ABB RAPID module: Module1.mod

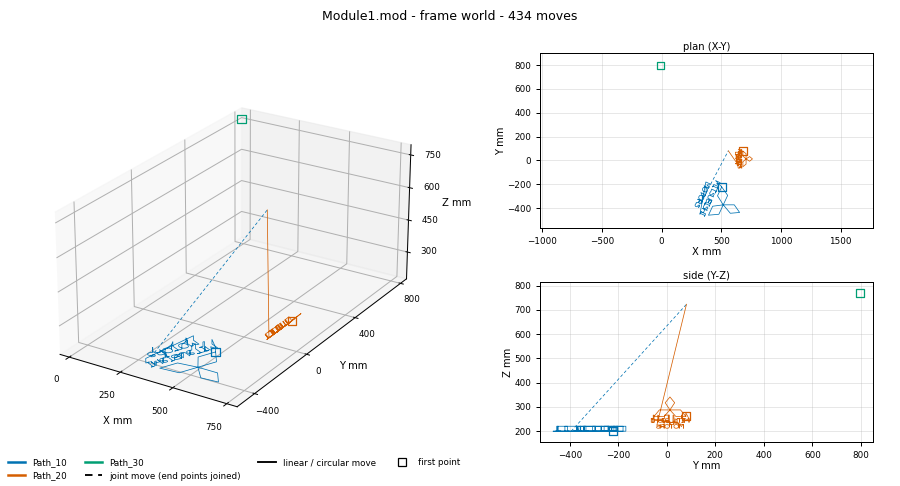
[picture p0: tool path of Module1.mod in frame world, 434 of 434 moves have a stored position in this frame; points joined in program order, loops and branches not executed]
MODULE Module1
    PERS tooldata TCP:=[TRUE,[[-35.118,-0.77,114.286],[1,0,0,0]],[1,[0,0,1],[1,0,0,0],0,0,0]];
    TASK PERS wobjdata Workobject_5:=[FALSE,TRUE,"",[[411.94279579,7.766562071,169.6],[0.537299678,0,0,-0.843391401]],[[0,0,30],[1,0,0,0]]];
    TASK PERS wobjdata Workobject_6:=[FALSE,TRUE,"",[[628.009,163.117,186.516],[0.653281027,0.27059915,-0.27059915,-0.653281027]],[[0,0,15],[1,0,0,0]]];

    CONST robtarget Target_4030:=[[169.057210378,179.421981942,0],[0,0.923879533,-0.382683432,0],[0, 0, 0, 0],[9E+09,9E+09,9E+09,9E+09,9E+09,9E+09]];
    CONST robtarget Target_4040:=[[212.704790581,255.022303499,0],[0,0.923879533,-0.382683432,0],[0, 0, 0, 0],[9E+09,9E+09,9E+09,9E+09,9E+09,9E+09]];
    CONST robtarget Target_4050:=[[387.295111711,255.022303682,0],[0,0.923879533,-0.382683432,0],[0, 0, 0, 0],[9E+09,9E+09,9E+09,9E+09,9E+09,9E+09]];
    CONST robtarget Target_4060:=[[430.942692072,179.421982217,0],[0,0.923879533,-0.382683432,0],[0, 0, 0, 0],[9E+09,9E+09,9E+09,9E+09,9E+09,9E+09]];
    CONST robtarget Target_4070:=[[348.163115412,179.42198213,0],[0,0.923879533,-0.382683432,0],[0, 0, 0, 0],[9E+09,9E+09,9E+09,9E+09,9E+09,9E+09]];
    CONST robtarget Target_4080:=[[299.999951146,255.02230359,0],[0,0.923879533,-0.382683432,0],[0, 0, 0, 0],[9E+09,9E+09,9E+09,9E+09,9E+09,9E+09]];
    CONST robtarget Target_4090:=[[260.995941008,338.665964696,0],[0,0.923879533,-0.382683432,0],[0, 0, 0, 0],[9E+09,9E+09,9E+09,9E+09,9E+09,9E+09]];
    CONST robtarget Target_4100:=[[299.999950987,406.221532398,0],[0,0.923879533,-0.382683432,0],[0, 0, 0, 0],[9E+09,9E+09,9E+09,9E+09,9E+09,9E+09]];
    CONST robtarget Target_4110:=[[339.003961108,338.665964778,0],[0,0.923879533,-0.382683432,0],[0, 0, 0, 0],[9E+09,9E+09,9E+09,9E+09,9E+09,9E+09]];
    CONST robtarget Target_4120:=[[299.999951146,255.02230359,0],[0,0.923879533,-0.382683432,0],[0, 0, 0, 0],[9E+09,9E+09,9E+09,9E+09,9E+09,9E+09]];
    CONST robtarget Target_4130:=[[251.837494145,179.422689136,0],[0,0.923879533,-0.382683432,0],[0, 0, 0, 0],[9E+09,9E+09,9E+09,9E+09,9E+09,9E+09]];
    CONST robtarget Target_4140:=[[169.057210378,179.421981942,0],[0,0.923879533,-0.382683432,0],[0, 0, 0, 0],[9E+09,9E+09,9E+09,9E+09,9E+09,9E+09]];
    CONST robtarget Target_4150:=[[169.057210378,179.421981942,20.4],[0,0.923879533,-0.382683432,0],[0, 0, 0, 0],[9E+09,9E+09,9E+09,9E+09,9E+09,9E+09]];
    CONST robtarget Target_4160:=[[142.914058536,110.942932798,20.4],[0,0.923879533,-0.382683432,0],[0, 0, 0, 0],[9E+09,9E+09,9E+09,9E+09,9E+09,9E+09]];
    CONST robtarget Target_4170:=[[142.914058536,110.942932798,0],[0,0.923879533,-0.382683432,0],[0, 0, 0, 0],[9E+09,9E+09,9E+09,9E+09,9E+09,9E+09]];
    CONST robtarget Target_4180:=[[142.914058492,152.942247173,0],[0,0.923879533,-0.382683432,0],[0, 0, 0, 0],[9E+09,9E+09,9E+09,9E+09,9E+09,9E+09]];
    CONST robtarget Target_4190:=[[150.538083807,152.942247181,0],[0,0.923879533,-0.382683432,0],[0, 0, 0, 0],[9E+09,9E+09,9E+09,9E+09,9E+09,9E+09]];
    CONST robtarget Target_4200:=[[161.020941862,129.560347259,0],[0,0.923879533,-0.382683432,0],[0, 0, 0, 0],[9E+09,9E+09,9E+09,9E+09,9E+09,9E+09]];
    CONST robtarget Target_4210:=[[171.163681507,152.942954309,0],[0,0.923879533,-0.382683432,0],[0, 0, 0, 0],[9E+09,9E+09,9E+09,9E+09,9E+09,9E+09]];
    CONST robtarget Target_4220:=[[178.923471324,152.942954318,0],[0,0.923879533,-0.382683432,0],[0, 0, 0, 0],[9E+09,9E+09,9E+09,9E+09,9E+09,9E+09]];
    CONST robtarget Target_4230:=[[178.923471368,110.942225729,0],[0,0.923879533,-0.382683432,0],[0, 0, 0, 0],[9E+09,9E+09,9E+09,9E+09,9E+09,9E+09]];
    CONST robtarget Target_4240:=[[178.923471368,110.942225729,20.4],[0,0.923879533,-0.382683432,0],[0, 0, 0, 0],[9E+09,9E+09,9E+09,9E+09,9E+09,9E+09]];
    CONST robtarget Target_4250:=[[185.798670601,110.942932843,20.4],[0,0.923879533,-0.382683432,0],[0, 0, 0, 0],[9E+09,9E+09,9E+09,9E+09,9E+09,9E+09]];
    CONST robtarget Target_4260:=[[185.798670601,110.942932843,0],[0,0.923879533,-0.382683432,0],[0, 0, 0, 0],[9E+09,9E+09,9E+09,9E+09,9E+09,9E+09]];
    CONST robtarget Target_4270:=[[202.067783423,110.94293286,0],[0,0.923879533,-0.382683432,0],[0, 0, 0, 0],[9E+09,9E+09,9E+09,9E+09,9E+09,9E+09]];
    CONST robtarget Target_4280:=[[193.933227012,110.942932851,0],[0,0.923879533,-0.382683432,0],[0, 0, 0, 0],[9E+09,9E+09,9E+09,9E+09,9E+09,9E+09]];
    CONST robtarget Target_4290:=[[193.933226968,152.942247227,0],[0,0.923879533,-0.382683432,0],[0, 0, 0, 0],[9E+09,9E+09,9E+09,9E+09,9E+09,9E+09]];
    CONST robtarget Target_4300:=[[185.798670557,152.942247218,0],[0,0.923879533,-0.382683432,0],[0, 0, 0, 0],[9E+09,9E+09,9E+09,9E+09,9E+09,9E+09]];
    CONST robtarget Target_4310:=[[202.067783379,152.942247235,0],[0,0.923879533,-0.382683432,0],[0, 0, 0, 0],[9E+09,9E+09,9E+09,9E+09,9E+09,9E+09]];
    CONST robtarget Target_4320:=[[202.067783379,152.942247235,20.4],[0,0.923879533,-0.382683432,0],[0, 0, 0, 0],[9E+09,9E+09,9E+09,9E+09,9E+09,9E+09]];
    CONST robtarget Target_4330:=[[204.689028217,152.942954345,20.4],[0,0.923879533,-0.382683432,0],[0, 0, 0, 0],[9E+09,9E+09,9E+09,9E+09,9E+09,9E+09]];
    CONST robtarget Target_4340:=[[204.689028217,152.942954345,0],[0,0.923879533,-0.382683432,0],[0, 0, 0, 0],[9E+09,9E+09,9E+09,9E+09,9E+09,9E+09]];
    CONST robtarget Target_4350:=[[238.451962805,152.94295438,0],[0,0.923879533,-0.382683432,0],[0, 0, 0, 0],[9E+09,9E+09,9E+09,9E+09,9E+09,9E+09]];
    CONST robtarget Target_4360:=[[221.570495511,152.942954362,0],[0,0.923879533,-0.382683432,0],[0, 0, 0, 0],[9E+09,9E+09,9E+09,9E+09,9E+09,9E+09]];
    CONST robtarget Target_4370:=[[221.570495555,110.942225773,0],[0,0.923879533,-0.382683432,0],[0, 0, 0, 0],[9E+09,9E+09,9E+09,9E+09,9E+09,9E+09]];
    CONST robtarget Target_4380:=[[221.570495555,110.942225773,20.4],[0,0.923879533,-0.382683432,0],[0, 0, 0, 0],[9E+09,9E+09,9E+09,9E+09,9E+09,9E+09]];
    CONST robtarget Target_4390:=[[240.630558839,113.461647255,20.4],[0,0.923879533,-0.382683432,0],[0, 0, 0, 0],[9E+09,9E+09,9E+09,9E+09,9E+09,9E+09]];
    CONST robtarget Target_4400:=[[240.630558839,113.461647255,0],[0,0.923879533,-0.382683432,0],[0, 0, 0, 0],[9E+09,9E+09,9E+09,9E+09,9E+09,9E+09]];
    CONST robtarget Target_4410:=[[254.414898435,110.193399727,0],[0,0.923879533,-0.382683432,0],[0, 0, 0, 0],[9E+09,9E+09,9E+09,9E+09,9E+09,9E+09]];
    CONST robtarget Target_4420:=[[260.813507697,111.181227907,0],[0,0.923879533,-0.382683432,0],[0, 0, 0, 0],[9E+09,9E+09,9E+09,9E+09,9E+09,9E+09]];
    CONST robtarget Target_4430:=[[265.374346433,114.005412395,0],[0,0.923879533,-0.382683432,0],[0, 0, 0, 0],[9E+09,9E+09,9E+09,9E+09,9E+09,9E+09]];
    CONST robtarget Target_4440:=[[268.182267456,118.056427148,0],[0,0.923879533,-0.382683432,0],[0, 0, 0, 0],[9E+09,9E+09,9E+09,9E+09,9E+09,9E+09]];
    CONST robtarget Target_4450:=[[269.186359081,122.922736017,0],[0,0.923879533,-0.382683432,0],[0, 0, 0, 0],[9E+09,9E+09,9E+09,9E+09,9E+09,9E+09]];
    CONST robtarget Target_4460:=[[267.178175815,129.508728575,0],[0,0.923879533,-0.382683432,0],[0, 0, 0, 0],[9E+09,9E+09,9E+09,9E+09,9E+09,9E+09]];
    CONST robtarget Target_4470:=[[260.847448799,133.508831629,0],[0,0.923879533,-0.382683432,0],[0, 0, 0, 0],[9E+09,9E+09,9E+09,9E+09,9E+09,9E+09]];
    CONST robtarget Target_4480:=[[256.575816733,134.631010087,0],[0,0.923879533,-0.382683432,0],[0, 0, 0, 0],[9E+09,9E+09,9E+09,9E+09,9E+09,9E+09]];
    CONST robtarget Target_4490:=[[252.236302415,135.720661632,0],[0,0.923879533,-0.382683432,0],[0, 0, 0, 0],[9E+09,9E+09,9E+09,9E+09,9E+09,9E+09]];
    CONST robtarget Target_4500:=[[248.169731314,138.01805156,0],[0,0.923879533,-0.382683432,0],[0, 0, 0, 0],[9E+09,9E+09,9E+09,9E+09,9E+09,9E+09]];
    CONST robtarget Target_4510:=[[246.756931961,142.255035391,0],[0,0.923879533,-0.382683432,0],[0, 0, 0, 0],[9E+09,9E+09,9E+09,9E+09,9E+09,9E+09]];
    CONST robtarget Target_4520:=[[249.156145265,147.037198555,0],[0,0.923879533,-0.382683432,0],[0, 0, 0, 0],[9E+09,9E+09,9E+09,9E+09,9E+09,9E+09]];
    CONST robtarget Target_4530:=[[255.435960587,148.857998523,0],[0,0.923879533,-0.382683432,0],[0, 0, 0, 0],[9E+09,9E+09,9E+09,9E+09,9E+09,9E+09]];
    CONST robtarget Target_4540:=[[262.004275478,147.496817976,0],[0,0.923879533,-0.382683432,0],[0, 0, 0, 0],[9E+09,9E+09,9E+09,9E+09,9E+09,9E+09]];
    CONST robtarget Target_4550:=[[267.144234674,144.297159797,0],[0,0.923879533,-0.382683432,0],[0, 0, 0, 0],[9E+09,9E+09,9E+09,9E+09,9E+09,9E+09]];
    CONST robtarget Target_4560:=[[267.144234674,144.297159797,20.4],[0,0.923879533,-0.382683432,0],[0, 0, 0, 0],[9E+09,9E+09,9E+09,9E+09,9E+09,9E+09]];
    CONST robtarget Target_4570:=[[274.35955226,152.942247311,20.4],[0,0.923879533,-0.382683432,0],[0, 0, 0, 0],[9E+09,9E+09,9E+09,9E+09,9E+09,9E+09]];
    CONST robtarget Target_4580:=[[274.35955226,152.942247311,0],[0,0.923879533,-0.382683432,0],[0, 0, 0, 0],[9E+09,9E+09,9E+09,9E+09,9E+09,9E+09]];
    CONST robtarget Target_4590:=[[274.360259381,139.838851549,0],[0,0.923879533,-0.382683432,0],[0, 0, 0, 0],[9E+09,9E+09,9E+09,9E+09,9E+09,9E+09]];
    CONST robtarget Target_4600:=[[274.359552288,126.735455787,0],[0,0.923879533,-0.382683432,0],[0, 0, 0, 0],[9E+09,9E+09,9E+09,9E+09,9E+09,9E+09]];
    CONST robtarget Target_4610:=[[275.261820549,119.179312724,0],[0,0.923879533,-0.382683432,0],[0, 0, 0, 0],[9E+09,9E+09,9E+09,9E+09,9E+09,9E+09]];
    CONST robtarget Target_4620:=[[278.375918818,113.938237265,0],[0,0.923879533,-0.382683432,0],[0, 0, 0, 0],[9E+09,9E+09,9E+09,9E+09,9E+09,9E+09]];
    CONST robtarget Target_4630:=[[283.072522062,111.027785758,0],[0,0.923879533,-0.382683432,0],[0, 0, 0, 0],[9E+09,9E+09,9E+09,9E+09,9E+09,9E+09]];
    CONST robtarget Target_4640:=[[289.539720684,110.057635261,0],[0,0.923879533,-0.382683432,0],[0, 0, 0, 0],[9E+09,9E+09,9E+09,9E+09,9E+09,9E+09]];
    CONST robtarget Target_4650:=[[296.074801555,111.010815209,0],[0,0.923879533,-0.382683432,0],[0, 0, 0, 0],[9E+09,9E+09,9E+09,9E+09,9E+09,9E+09]];
    CONST robtarget Target_4660:=[[300.737463667,113.938237288,0],[0,0.923879533,-0.382683432,0],[0, 0, 0, 0],[9E+09,9E+09,9E+09,9E+09,9E+09,9E+09]];
    CONST robtarget Target_4670:=[[303.868532488,119.213253879,0],[0,0.923879533,-0.382683432,0],[0, 0, 0, 0],[9E+09,9E+09,9E+09,9E+09,9E+09,9E+09]];
    CONST robtarget Target_4680:=[[304.75383017,126.735455818,0],[0,0.923879533,-0.382683432,0],[0, 0, 0, 0],[9E+09,9E+09,9E+09,9E+09,9E+09,9E+09]];
    CONST robtarget Target_4690:=[[304.75312305,139.838851581,0],[0,0.923879533,-0.382683432,0],[0, 0, 0, 0],[9E+09,9E+09,9E+09,9E+09,9E+09,9E+09]];
    CONST robtarget Target_4700:=[[304.753830143,152.942247343,0],[0,0.923879533,-0.382683432,0],[0, 0, 0, 0],[9E+09,9E+09,9E+09,9E+09,9E+09,9E+09]];
    CONST robtarget Target_4710:=[[304.753830143,152.942247343,20.4],[0,0.923879533,-0.382683432,0],[0, 0, 0, 0],[9E+09,9E+09,9E+09,9E+09,9E+09,9E+09]];
    CONST robtarget Target_4720:=[[312.751914945,152.942954458,20.4],[0,0.923879533,-0.382683432,0],[0, 0, 0, 0],[9E+09,9E+09,9E+09,9E+09,9E+09,9E+09]];
    CONST robtarget Target_4730:=[[312.751914945,152.942954458,0],[0,0.923879533,-0.382683432,0],[0, 0, 0, 0],[9E+09,9E+09,9E+09,9E+09,9E+09,9E+09]];
    CONST robtarget Target_4740:=[[312.751914989,110.942225869,0],[0,0.923879533,-0.382683432,0],[0, 0, 0, 0],[9E+09,9E+09,9E+09,9E+09,9E+09,9E+09]];
    CONST robtarget Target_4750:=[[318.776464765,110.942225875,0],[0,0.923879533,-0.382683432,0],[0, 0, 0, 0],[9E+09,9E+09,9E+09,9E+09,9E+09,9E+09]];
    CONST robtarget Target_4760:=[[324.800307434,110.942932988,0],[0,0.923879533,-0.382683432,0],[0, 0, 0, 0],[9E+09,9E+09,9E+09,9E+09,9E+09,9E+09]];
    CONST robtarget Target_4770:=[[331.795007712,111.724993096,0],[0,0.923879533,-0.382683432,0],[0, 0, 0, 0],[9E+09,9E+09,9E+09,9E+09,9E+09,9E+09]];
    CONST robtarget Target_4780:=[[336.882641,114.346237939,0],[0,0.923879533,-0.382683432,0],[0, 0, 0, 0],[9E+09,9E+09,9E+09,9E+09,9E+09,9E+09]];
    CONST robtarget Target_4790:=[[340.048358055,118.310985664,0],[0,0.923879533,-0.382683432,0],[0, 0, 0, 0],[9E+09,9E+09,9E+09,9E+09,9E+09,9E+09]];
    CONST robtarget Target_4800:=[[341.239832976,123.842682015,0],[0,0.923879533,-0.382683432,0],[0, 0, 0, 0],[9E+09,9E+09,9E+09,9E+09,9E+09,9E+09]];
    CONST robtarget Target_4810:=[[339.180738022,130.564439075,0],[0,0.923879533,-0.382683432,0],[0, 0, 0, 0],[9E+09,9E+09,9E+09,9E+09,9E+09,9E+09]];
    CONST robtarget Target_4820:=[[333.377512665,134.495245665,0],[0,0.923879533,-0.382683432,0],[0, 0, 0, 0],[9E+09,9E+09,9E+09,9E+09,9E+09,9E+09]];
    CONST robtarget Target_4830:=[[312.751914967,131.94329727,0],[0,0.923879533,-0.382683432,0],[0, 0, 0, 0],[9E+09,9E+09,9E+09,9E+09,9E+09,9E+09]];
    CONST robtarget Target_4840:=[[333.377512665,134.291598912,0],[0,0.923879533,-0.382683432,0],[0, 0, 0, 0],[9E+09,9E+09,9E+09,9E+09,9E+09,9E+09]];
    CONST robtarget Target_4850:=[[337.700056414,138.171493825,0],[0,0.923879533,-0.382683432,0],[0, 0, 0, 0],[9E+09,9E+09,9E+09,9E+09,9E+09,9E+09]];
    CONST robtarget Target_4860:=[[339.265590822,143.48045154,0],[0,0.923879533,-0.382683432,0],[0, 0, 0, 0],[9E+09,9E+09,9E+09,9E+09,9E+09,9E+09]];
    CONST robtarget Target_4870:=[[338.227558063,148.092201966,0],[0,0.923879533,-0.382683432,0],[0, 0, 0, 0],[9E+09,9E+09,9E+09,9E+09,9E+09,9E+09]];
    CONST robtarget Target_4880:=[[334.909105935,151.240948459,0],[0,0.923879533,-0.382683432,0],[0, 0, 0, 0],[9E+09,9E+09,9E+09,9E+09,9E+09,9E+09]];
    CONST robtarget Target_4890:=[[323.881775681,152.94295447,0],[0,0.923879533,-0.382683432,0],[0, 0, 0, 0],[9E+09,9E+09,9E+09,9E+09,9E+09,9E+09]];
    CONST robtarget Target_4900:=[[318.316845313,152.942954464,0],[0,0.923879533,-0.382683432,0],[0, 0, 0, 0],[9E+09,9E+09,9E+09,9E+09,9E+09,9E+09]];
    CONST robtarget Target_4910:=[[312.751914945,152.942954458,0],[0,0.923879533,-0.382683432,0],[0, 0, 0, 0],[9E+09,9E+09,9E+09,9E+09,9E+09,9E+09]];
    CONST robtarget Target_4920:=[[312.751914945,152.942954458,20.4],[0,0.923879533,-0.382683432,0],[0, 0, 0, 0],[9E+09,9E+09,9E+09,9E+09,9E+09,9E+09]];
    CONST robtarget Target_4930:=[[345.153668979,152.942247385,20.4],[0,0.923879533,-0.382683432,0],[0, 0, 0, 0],[9E+09,9E+09,9E+09,9E+09,9E+09,9E+09]];
    CONST robtarget Target_4940:=[[345.153668979,152.942247385,0],[0,0.923879533,-0.382683432,0],[0, 0, 0, 0],[9E+09,9E+09,9E+09,9E+09,9E+09,9E+09]];
    CONST robtarget Target_4950:=[[361.422781801,152.942247402,0],[0,0.923879533,-0.382683432,0],[0, 0, 0, 0],[9E+09,9E+09,9E+09,9E+09,9E+09,9E+09]];
    CONST robtarget Target_4960:=[[353.28822539,152.942247394,0],[0,0.923879533,-0.382683432,0],[0, 0, 0, 0],[9E+09,9E+09,9E+09,9E+09,9E+09,9E+09]];
    CONST robtarget Target_4970:=[[353.288225434,110.942933018,0],[0,0.923879533,-0.382683432,0],[0, 0, 0, 0],[9E+09,9E+09,9E+09,9E+09,9E+09,9E+09]];
    CONST robtarget Target_4980:=[[345.153669023,110.94293301,0],[0,0.923879533,-0.382683432,0],[0, 0, 0, 0],[9E+09,9E+09,9E+09,9E+09,9E+09,9E+09]];
    CONST robtarget Target_4990:=[[361.422781845,110.942933027,0],[0,0.923879533,-0.382683432,0],[0, 0, 0, 0],[9E+09,9E+09,9E+09,9E+09,9E+09,9E+09]];
    CONST robtarget Target_5000:=[[361.422781845,110.942933027,20.4],[0,0.923879533,-0.382683432,0],[0, 0, 0, 0],[9E+09,9E+09,9E+09,9E+09,9E+09,9E+09]];
    CONST robtarget Target_5010:=[[356.079175895,115.231535649,0],[0,0.923879533,-0.382683432,0],[0, 0, 0, 0],[9E+09,9E+09,9E+09,9E+09,9E+09,9E+09]];
    CONST robtarget Target_5020:=[[366.255856692,113.46094028,20.4],[0,0.923879533,-0.382683432,0],[0, 0, 0, 0],[9E+09,9E+09,9E+09,9E+09,9E+09,9E+09]];
    CONST robtarget Target_5030:=[[366.255856692,113.46094028,0],[0,0.923879533,-0.382683432,0],[0, 0, 0, 0],[9E+09,9E+09,9E+09,9E+09,9E+09,9E+09]];
    CONST robtarget Target_5040:=[[380.040196287,110.194106965,0],[0,0.923879533,-0.382683432,0],[0, 0, 0, 0],[9E+09,9E+09,9E+09,9E+09,9E+09,9E+09]];
    CONST robtarget Target_5050:=[[386.438805549,111.180520932,0],[0,0.923879533,-0.382683432,0],[0, 0, 0, 0],[9E+09,9E+09,9E+09,9E+09,9E+09,9E+09]];
    CONST robtarget Target_5060:=[[390.999644285,114.006119634,0],[0,0.923879533,-0.382683432,0],[0, 0, 0, 0],[9E+09,9E+09,9E+09,9E+09,9E+09,9E+09]];
    CONST robtarget Target_5070:=[[393.807565309,118.055720173,0],[0,0.923879533,-0.382683432,0],[0, 0, 0, 0],[9E+09,9E+09,9E+09,9E+09,9E+09,9E+09]];
    CONST robtarget Target_5080:=[[394.811656933,122.923443255,0],[0,0.923879533,-0.382683432,0],[0, 0, 0, 0],[9E+09,9E+09,9E+09,9E+09,9E+09,9E+09]];
    CONST robtarget Target_5090:=[[392.803473668,129.509435813,0],[0,0.923879533,-0.382683432,0],[0, 0, 0, 0],[9E+09,9E+09,9E+09,9E+09,9E+09,9E+09]];
    CONST robtarget Target_5100:=[[386.472746651,133.508124654,0],[0,0.923879533,-0.382683432,0],[0, 0, 0, 0],[9E+09,9E+09,9E+09,9E+09,9E+09,9E+09]];
    CONST robtarget Target_5110:=[[382.201821692,134.631010218,0],[0,0.923879533,-0.382683432,0],[0, 0, 0, 0],[9E+09,9E+09,9E+09,9E+09,9E+09,9E+09]];
    CONST robtarget Target_5120:=[[377.862307375,135.720661764,0],[0,0.923879533,-0.382683432,0],[0, 0, 0, 0],[9E+09,9E+09,9E+09,9E+09,9E+09,9E+09]];
    CONST robtarget Target_5130:=[[373.79432206,138.018051691,0],[0,0.923879533,-0.382683432,0],[0, 0, 0, 0],[9E+09,9E+09,9E+09,9E+09,9E+09,9E+09]];
    CONST robtarget Target_5140:=[[372.382229814,142.25574263,0],[0,0.923879533,-0.382683432,0],[0, 0, 0, 0],[9E+09,9E+09,9E+09,9E+09,9E+09,9E+09]];
    CONST robtarget Target_5150:=[[374.782150224,147.037198687,0],[0,0.923879533,-0.382683432,0],[0, 0, 0, 0],[9E+09,9E+09,9E+09,9E+09,9E+09,9E+09]];
    CONST robtarget Target_5160:=[[381.061258439,148.858705761,0],[0,0.923879533,-0.382683432,0],[0, 0, 0, 0],[9E+09,9E+09,9E+09,9E+09,9E+09,9E+09]];
    CONST robtarget Target_5170:=[[387.630280438,147.496818108,0],[0,0.923879533,-0.382683432,0],[0, 0, 0, 0],[9E+09,9E+09,9E+09,9E+09,9E+09,9E+09]];
    CONST robtarget Target_5180:=[[392.769532527,144.297867035,0],[0,0.923879533,-0.382683432,0],[0, 0, 0, 0],[9E+09,9E+09,9E+09,9E+09,9E+09,9E+09]];
    CONST robtarget Target_5190:=[[392.769532527,144.297867035,20.4],[0,0.923879533,-0.382683432,0],[0, 0, 0, 0],[9E+09,9E+09,9E+09,9E+09,9E+09,9E+09]];
    CONST robtarget Target_5200:=[[400.496088316,152.942247443,20.4],[0,0.923879533,-0.382683432,0],[0, 0, 0, 0],[9E+09,9E+09,9E+09,9E+09,9E+09,9E+09]];
    CONST robtarget Target_5210:=[[400.496088316,152.942247443,0],[0,0.923879533,-0.382683432,0],[0, 0, 0, 0],[9E+09,9E+09,9E+09,9E+09,9E+09,9E+09]];
    CONST robtarget Target_5220:=[[400.49608836,110.942933068,0],[0,0.923879533,-0.382683432,0],[0, 0, 0, 0],[9E+09,9E+09,9E+09,9E+09,9E+09,9E+09]];
    CONST robtarget Target_5230:=[[400.496088338,131.942590255,0],[0,0.923879533,-0.382683432,0],[0, 0, 0, 0],[9E+09,9E+09,9E+09,9E+09,9E+09,9E+09]];
    CONST robtarget Target_5240:=[[430.992189597,131.942590287,0],[0,0.923879533,-0.382683432,0],[0, 0, 0, 0],[9E+09,9E+09,9E+09,9E+09,9E+09,9E+09]];
    CONST robtarget Target_5250:=[[430.991482512,110.942225993,0],[0,0.923879533,-0.382683432,0],[0, 0, 0, 0],[9E+09,9E+09,9E+09,9E+09,9E+09,9E+09]];
    CONST robtarget Target_5260:=[[430.991482468,152.942954582,0],[0,0.923879533,-0.382683432,0],[0, 0, 0, 0],[9E+09,9E+09,9E+09,9E+09,9E+09,9E+09]];
    CONST robtarget Target_5270:=[[430.991482468,152.942954582,20.4],[0,0.923879533,-0.382683432,0],[0, 0, 0, 0],[9E+09,9E+09,9E+09,9E+09,9E+09,9E+09]];
    CONST robtarget Target_5280:=[[437.866681701,152.942247482,20.4],[0,0.923879533,-0.382683432,0],[0, 0, 0, 0],[9E+09,9E+09,9E+09,9E+09,9E+09,9E+09]];
    CONST robtarget Target_5290:=[[437.866681701,152.942247482,0],[0,0.923879533,-0.382683432,0],[0, 0, 0, 0],[9E+09,9E+09,9E+09,9E+09,9E+09,9E+09]];
    CONST robtarget Target_5300:=[[454.135794523,152.942247499,0],[0,0.923879533,-0.382683432,0],[0, 0, 0, 0],[9E+09,9E+09,9E+09,9E+09,9E+09,9E+09]];
    CONST robtarget Target_5310:=[[446.001238112,152.942247491,0],[0,0.923879533,-0.382683432,0],[0, 0, 0, 0],[9E+09,9E+09,9E+09,9E+09,9E+09,9E+09]];
    CONST robtarget Target_5320:=[[446.001238156,110.942933116,0],[0,0.923879533,-0.382683432,0],[0, 0, 0, 0],[9E+09,9E+09,9E+09,9E+09,9E+09,9E+09]];
    CONST robtarget Target_5330:=[[437.866681745,110.942933107,0],[0,0.923879533,-0.382683432,0],[0, 0, 0, 0],[9E+09,9E+09,9E+09,9E+09,9E+09,9E+09]];
    CONST robtarget Target_5340:=[[454.135794567,110.942933124,0],[0,0.923879533,-0.382683432,0],[0, 0, 0, 0],[9E+09,9E+09,9E+09,9E+09,9E+09,9E+09]];
    CONST robtarget Target_5350:=[[454.135794567,110.942933124,20.4],[0,0.923879533,-0.382683432,0],[0, 0, 0, 0],[9E+09,9E+09,9E+09,9E+09,9E+09,9E+09]];
    CONST robtarget Target_5360:=[[187.97655956,41.790718072,20.4],[0,0.923879533,-0.382683432,0],[0, 0, 0, 0],[9E+09,9E+09,9E+09,9E+09,9E+09,9E+09]];
    CONST robtarget Target_5370:=[[187.97655956,41.790718072,0],[0,0.923879533,-0.382683432,0],[0, 0, 0, 0],[9E+09,9E+09,9E+09,9E+09,9E+09,9E+09]];
    CONST robtarget Target_5380:=[[187.977266623,83.790739554,0],[0,0.923879533,-0.382683432,0],[0, 0, 0, 0],[9E+09,9E+09,9E+09,9E+09,9E+09,9E+09]];
    CONST robtarget Target_5390:=[[195.601291938,83.790739562,0],[0,0.923879533,-0.382683432,0],[0, 0, 0, 0],[9E+09,9E+09,9E+09,9E+09,9E+09,9E+09]];
    CONST robtarget Target_5400:=[[206.084149993,60.40883964,0],[0,0.923879533,-0.382683432,0],[0, 0, 0, 0],[9E+09,9E+09,9E+09,9E+09,9E+09,9E+09]];
    CONST robtarget Target_5410:=[[216.226182531,83.790739584,0],[0,0.923879533,-0.382683432,0],[0, 0, 0, 0],[9E+09,9E+09,9E+09,9E+09,9E+09,9E+09]];
    CONST robtarget Target_5420:=[[223.987386561,83.790739592,0],[0,0.923879533,-0.382683432,0],[0, 0, 0, 0],[9E+09,9E+09,9E+09,9E+09,9E+09,9E+09]];
    CONST robtarget Target_5430:=[[223.986679499,41.79071811,0],[0,0.923879533,-0.382683432,0],[0, 0, 0, 0],[9E+09,9E+09,9E+09,9E+09,9E+09,9E+09]];
    CONST robtarget Target_5440:=[[223.986679499,41.79071811,20.4],[0,0.923879533,-0.382683432,0],[0, 0, 0, 0],[9E+09,9E+09,9E+09,9E+09,9E+09,9E+09]];
    CONST robtarget Target_5450:=[[230.113052629,62.790375304,20.4],[0,0.923879533,-0.382683432,0],[0, 0, 0, 0],[9E+09,9E+09,9E+09,9E+09,9E+09,9E+09]];
    CONST robtarget Target_5460:=[[230.113052629,62.790375304,0],[0,0.923879533,-0.382683432,0],[0, 0, 0, 0],[9E+09,9E+09,9E+09,9E+09,9E+09,9E+09]];
    CONST robtarget Target_5470:=[[231.407058048,53.515962763,0],[0,0.923879533,-0.382683432,0],[0, 0, 0, 0],[9E+09,9E+09,9E+09,9E+09,9E+09,9E+09]];
    CONST robtarget Target_5480:=[[235.117247336,46.623792971,0],[0,0.923879533,-0.382683432,0],[0, 0, 0, 0],[9E+09,9E+09,9E+09,9E+09,9E+09,9E+09]];
    CONST robtarget Target_5490:=[[241.004618401,42.352868019,0],[0,0.923879533,-0.382683432,0],[0, 0, 0, 0],[9E+09,9E+09,9E+09,9E+09,9E+09,9E+09]];
    CONST robtarget Target_5500:=[[248.662584843,40.906127552,0],[0,0.923879533,-0.382683432,0],[0, 0, 0, 0],[9E+09,9E+09,9E+09,9E+09,9E+09,9E+09]];
    CONST robtarget Target_5510:=[[256.201050235,42.30124924,0],[0,0.923879533,-0.382683432,0],[0, 0, 0, 0],[9E+09,9E+09,9E+09,9E+09,9E+09,9E+09]];
    CONST robtarget Target_5520:=[[262.209336551,46.623792999,0],[0,0.923879533,-0.382683432,0],[0, 0, 0, 0],[9E+09,9E+09,9E+09,9E+09,9E+09,9E+09]];
    CONST robtarget Target_5530:=[[265.952759843,53.550611032,0],[0,0.923879533,-0.382683432,0],[0, 0, 0, 0],[9E+09,9E+09,9E+09,9E+09,9E+09,9E+09]];
    CONST robtarget Target_5540:=[[267.246058136,62.790375343,0],[0,0.923879533,-0.382683432,0],[0, 0, 0, 0],[9E+09,9E+09,9E+09,9E+09,9E+09,9E+09]];
    CONST robtarget Target_5550:=[[265.918818698,72.116406679,0],[0,0.923879533,-0.382683432,0],[0, 0, 0, 0],[9E+09,9E+09,9E+09,9E+09,9E+09,9E+09]];
    CONST robtarget Target_5560:=[[262.20862941,78.991605908,0],[0,0.923879533,-0.382683432,0],[0, 0, 0, 0],[9E+09,9E+09,9E+09,9E+09,9E+09,9E+09]];
    CONST robtarget Target_5570:=[[256.38843349,83.178385153,0],[0,0.923879533,-0.382683432,0],[0, 0, 0, 0],[9E+09,9E+09,9E+09,9E+09,9E+09,9E+09]];
    CONST robtarget Target_5580:=[[248.662584797,84.676037308,0],[0,0.923879533,-0.382683432,0],[0, 0, 0, 0],[9E+09,9E+09,9E+09,9E+09,9E+09,9E+09]];
    CONST robtarget Target_5590:=[[241.021588921,83.229296826,0],[0,0.923879533,-0.382683432,0],[0, 0, 0, 0],[9E+09,9E+09,9E+09,9E+09,9E+09,9E+09]];
    CONST robtarget Target_5600:=[[235.150481321,78.99160588,0],[0,0.923879533,-0.382683432,0],[0, 0, 0, 0],[9E+09,9E+09,9E+09,9E+09,9E+09,9E+09]];
    CONST robtarget Target_5610:=[[231.423321485,72.082465517,0],[0,0.923879533,-0.382683432,0],[0, 0, 0, 0],[9E+09,9E+09,9E+09,9E+09,9E+09,9E+09]];
    CONST robtarget Target_5620:=[[230.113052629,62.790375304,0],[0,0.923879533,-0.382683432,0],[0, 0, 0, 0],[9E+09,9E+09,9E+09,9E+09,9E+09,9E+09]];
    CONST robtarget Target_5630:=[[230.113052629,62.790375304,20.4],[0,0.923879533,-0.382683432,0],[0, 0, 0, 0],[9E+09,9E+09,9E+09,9E+09,9E+09,9E+09]];
    CONST robtarget Target_5640:=[[269.083828638,83.790739639,20.4],[0,0.923879533,-0.382683432,0],[0, 0, 0, 0],[9E+09,9E+09,9E+09,9E+09,9E+09,9E+09]];
    CONST robtarget Target_5650:=[[269.083828638,83.790739639,0],[0,0.923879533,-0.382683432,0],[0, 0, 0, 0],[9E+09,9E+09,9E+09,9E+09,9E+09,9E+09]];
    CONST robtarget Target_5660:=[[302.84817744,83.790739675,0],[0,0.923879533,-0.382683432,0],[0, 0, 0, 0],[9E+09,9E+09,9E+09,9E+09,9E+09,9E+09]];
    CONST robtarget Target_5670:=[[285.965295932,83.790739657,0],[0,0.923879533,-0.382683432,0],[0, 0, 0, 0],[9E+09,9E+09,9E+09,9E+09,9E+09,9E+09]];
    CONST robtarget Target_5680:=[[285.966003083,41.790718175,0],[0,0.923879533,-0.382683432,0],[0, 0, 0, 0],[9E+09,9E+09,9E+09,9E+09,9E+09,9E+09]];
    CONST robtarget Target_5690:=[[285.966003083,41.790718175,20.4],[0,0.923879533,-0.382683432,0],[0, 0, 0, 0],[9E+09,9E+09,9E+09,9E+09,9E+09,9E+09]];
    CONST robtarget Target_5700:=[[304.719182005,62.791082489,20.4],[0,0.923879533,-0.382683432,0],[0, 0, 0, 0],[9E+09,9E+09,9E+09,9E+09,9E+09,9E+09]];
    CONST robtarget Target_5710:=[[304.719182005,62.791082489,0],[0,0.923879533,-0.382683432,0],[0, 0, 0, 0],[9E+09,9E+09,9E+09,9E+09,9E+09,9E+09]];
    CONST robtarget Target_5720:=[[306.012480318,53.515962841,0],[0,0.923879533,-0.382683432,0],[0, 0, 0, 0],[9E+09,9E+09,9E+09,9E+09,9E+09,9E+09]];
    CONST robtarget Target_5730:=[[309.722669606,46.623793049,0],[0,0.923879533,-0.382683432,0],[0, 0, 0, 0],[9E+09,9E+09,9E+09,9E+09,9E+09,9E+09]];
    CONST robtarget Target_5740:=[[315.610747777,42.35216099,0],[0,0.923879533,-0.382683432,0],[0, 0, 0, 0],[9E+09,9E+09,9E+09,9E+09,9E+09,9E+09]];
    CONST robtarget Target_5750:=[[323.268714219,40.905420524,0],[0,0.923879533,-0.382683432,0],[0, 0, 0, 0],[9E+09,9E+09,9E+09,9E+09,9E+09,9E+09]];
    CONST robtarget Target_5760:=[[330.807886718,42.301249318,0],[0,0.923879533,-0.382683432,0],[0, 0, 0, 0],[9E+09,9E+09,9E+09,9E+09,9E+09,9E+09]];
    CONST robtarget Target_5770:=[[336.81475882,46.623793078,0],[0,0.923879533,-0.382683432,0],[0, 0, 0, 0],[9E+09,9E+09,9E+09,9E+09,9E+09,9E+09]];
    CONST robtarget Target_5780:=[[340.558889219,53.549904003,0],[0,0.923879533,-0.382683432,0],[0, 0, 0, 0],[9E+09,9E+09,9E+09,9E+09,9E+09,9E+09]];
    CONST robtarget Target_5790:=[[341.852187512,62.791082528,0],[0,0.923879533,-0.382683432,0],[0, 0, 0, 0],[9E+09,9E+09,9E+09,9E+09,9E+09,9E+09]];
    CONST robtarget Target_5800:=[[340.524948074,72.117113864,0],[0,0.923879533,-0.382683432,0],[0, 0, 0, 0],[9E+09,9E+09,9E+09,9E+09,9E+09,9E+09]];
    CONST robtarget Target_5810:=[[336.815465893,78.991605986,0],[0,0.923879533,-0.382683432,0],[0, 0, 0, 0],[9E+09,9E+09,9E+09,9E+09,9E+09,9E+09]];
    CONST robtarget Target_5820:=[[330.995269973,83.178385232,0],[0,0.923879533,-0.382683432,0],[0, 0, 0, 0],[9E+09,9E+09,9E+09,9E+09,9E+09,9E+09]];
    CONST robtarget Target_5830:=[[323.268714173,84.675330279,0],[0,0.923879533,-0.382683432,0],[0, 0, 0, 0],[9E+09,9E+09,9E+09,9E+09,9E+09,9E+09]];
    CONST robtarget Target_5840:=[[315.628425404,83.229296904,0],[0,0.923879533,-0.382683432,0],[0, 0, 0, 0],[9E+09,9E+09,9E+09,9E+09,9E+09,9E+09]];
    CONST robtarget Target_5850:=[[309.757317804,78.991605958,0],[0,0.923879533,-0.382683432,0],[0, 0, 0, 0],[9E+09,9E+09,9E+09,9E+09,9E+09,9E+09]];
    CONST robtarget Target_5860:=[[306.030157968,72.082465595,0],[0,0.923879533,-0.382683432,0],[0, 0, 0, 0],[9E+09,9E+09,9E+09,9E+09,9E+09,9E+09]];
    CONST robtarget Target_5870:=[[304.719182005,62.791082489,0],[0,0.923879533,-0.382683432,0],[0, 0, 0, 0],[9E+09,9E+09,9E+09,9E+09,9E+09,9E+09]];
    CONST robtarget Target_5880:=[[304.719182005,62.791082489,20.4],[0,0.923879533,-0.382683432,0],[0, 0, 0, 0],[9E+09,9E+09,9E+09,9E+09,9E+09,9E+09]];
    CONST robtarget Target_5890:=[[347.978560643,83.790739722,20.4],[0,0.923879533,-0.382683432,0],[0, 0, 0, 0],[9E+09,9E+09,9E+09,9E+09,9E+09,9E+09]];
    CONST robtarget Target_5900:=[[347.978560643,83.790739722,0],[0,0.923879533,-0.382683432,0],[0, 0, 0, 0],[9E+09,9E+09,9E+09,9E+09,9E+09,9E+09]];
    CONST robtarget Target_5910:=[[347.979267793,41.79071824,0],[0,0.923879533,-0.382683432,0],[0, 0, 0, 0],[9E+09,9E+09,9E+09,9E+09,9E+09,9E+09]];
    CONST robtarget Target_5920:=[[347.978560643,83.790739722,0],[0,0.923879533,-0.382683432,0],[0, 0, 0, 0],[9E+09,9E+09,9E+09,9E+09,9E+09,9E+09]];
    CONST robtarget Target_5930:=[[364.843764481,83.39970969,0],[0,0.923879533,-0.382683432,0],[0, 0, 0, 0],[9E+09,9E+09,9E+09,9E+09,9E+09,9E+09]];
    CONST robtarget Target_5940:=[[372.978320898,77.919632144,0],[0,0.923879533,-0.382683432,0],[0, 0, 0, 0],[9E+09,9E+09,9E+09,9E+09,9E+09,9E+09]];
    CONST robtarget Target_5950:=[[374.253941537,72.388642903,0],[0,0.923879533,-0.382683432,0],[0, 0, 0, 0],[9E+09,9E+09,9E+09,9E+09,9E+09,9E+09]];
    CONST robtarget Target_5960:=[[371.906347031,64.679764772,0],[0,0.923879533,-0.382683432,0],[0, 0, 0, 0],[9E+09,9E+09,9E+09,9E+09,9E+09,9E+09]];
    CONST robtarget Target_5970:=[[365.540971792,60.068014338,0],[0,0.923879533,-0.382683432,0],[0, 0, 0, 0],[9E+09,9E+09,9E+09,9E+09,9E+09,9E+09]];
    CONST robtarget Target_5980:=[[353.5604616,58.501772805,0],[0,0.923879533,-0.382683432,0],[0, 0, 0, 0],[9E+09,9E+09,9E+09,9E+09,9E+09,9E+09]];
    CONST robtarget Target_5990:=[[365.540971792,60.068014338,0],[0,0.923879533,-0.382683432,0],[0, 0, 0, 0],[9E+09,9E+09,9E+09,9E+09,9E+09,9E+09]];
    CONST robtarget Target_6000:=[[380.482845204,41.791425381,0],[0,0.923879533,-0.382683432,0],[0, 0, 0, 0],[9E+09,9E+09,9E+09,9E+09,9E+09,9E+09]];
    CONST robtarget Target_6010:=[[380.482845204,41.791425381,20.4],[0,0.923879533,-0.382683432,0],[0, 0, 0, 0],[9E+09,9E+09,9E+09,9E+09,9E+09,9E+09]];
    CONST robtarget Target_6020:=[[381.742202379,44.30943263,20.4],[0,0.923879533,-0.382683432,0],[0, 0, 0, 0],[9E+09,9E+09,9E+09,9E+09,9E+09,9E+09]];
    CONST robtarget Target_6030:=[[381.742202379,44.30943263,0],[0,0.923879533,-0.382683432,0],[0, 0, 0, 0],[9E+09,9E+09,9E+09,9E+09,9E+09,9E+09]];
    CONST robtarget Target_6040:=[[395.527249081,41.041892208,0],[0,0.923879533,-0.382683432,0],[0, 0, 0, 0],[9E+09,9E+09,9E+09,9E+09,9E+09,9E+09]];
    CONST robtarget Target_6050:=[[401.925151237,42.029013282,0],[0,0.923879533,-0.382683432,0],[0, 0, 0, 0],[9E+09,9E+09,9E+09,9E+09,9E+09,9E+09]];
    CONST robtarget Target_6060:=[[406.486697079,44.853904877,0],[0,0.923879533,-0.382683432,0],[0, 0, 0, 0],[9E+09,9E+09,9E+09,9E+09,9E+09,9E+09]];
    CONST robtarget Target_6070:=[[409.293910996,48.904212523,0],[0,0.923879533,-0.382683432,0],[0, 0, 0, 0],[9E+09,9E+09,9E+09,9E+09,9E+09,9E+09]];
    CONST robtarget Target_6080:=[[410.298709727,53.771228499,0],[0,0.923879533,-0.382683432,0],[0, 0, 0, 0],[9E+09,9E+09,9E+09,9E+09,9E+09,9E+09]];
    CONST robtarget Target_6090:=[[408.290526462,60.357221057,0],[0,0.923879533,-0.382683432,0],[0, 0, 0, 0],[9E+09,9E+09,9E+09,9E+09,9E+09,9E+09]];
    CONST robtarget Target_6100:=[[401.959092339,64.356617004,0],[0,0.923879533,-0.382683432,0],[0, 0, 0, 0],[9E+09,9E+09,9E+09,9E+09,9E+09,9E+09]];
    CONST robtarget Target_6110:=[[397.688167379,65.479502568,0],[0,0.923879533,-0.382683432,0],[0, 0, 0, 0],[9E+09,9E+09,9E+09,9E+09,9E+09,9E+09]];
    CONST robtarget Target_6120:=[[393.347945955,66.568447007,0],[0,0.923879533,-0.382683432,0],[0, 0, 0, 0],[9E+09,9E+09,9E+09,9E+09,9E+09,9E+09]];
    CONST robtarget Target_6130:=[[389.281374854,68.865836935,0],[0,0.923879533,-0.382683432,0],[0, 0, 0, 0],[9E+09,9E+09,9E+09,9E+09,9E+09,9E+09]];
    CONST robtarget Target_6140:=[[387.869282608,73.103527873,0],[0,0.923879533,-0.382683432,0],[0, 0, 0, 0],[9E+09,9E+09,9E+09,9E+09,9E+09,9E+09]];
    CONST robtarget Target_6150:=[[390.268495911,77.885691037,0],[0,0.923879533,-0.382683432,0],[0, 0, 0, 0],[9E+09,9E+09,9E+09,9E+09,9E+09,9E+09]];
    CONST robtarget Target_6160:=[[396.548311233,79.706491005,0],[0,0.923879533,-0.382683432,0],[0, 0, 0, 0],[9E+09,9E+09,9E+09,9E+09,9E+09,9E+09]];
    CONST robtarget Target_6170:=[[403.116626125,78.345310458,0],[0,0.923879533,-0.382683432,0],[0, 0, 0, 0],[9E+09,9E+09,9E+09,9E+09,9E+09,9E+09]];
    CONST robtarget Target_6180:=[[408.256585321,75.145652278,0],[0,0.923879533,-0.382683432,0],[0, 0, 0, 0],[9E+09,9E+09,9E+09,9E+09,9E+09,9E+09]];
    CONST robtarget HOME:=[[-128.642685613,102.00455871,523.17008013],[0.191341716,-0.800103145,0.331413574,0.461939766],[0, 0, 0, 0],[9E+09,9E+09,9E+09,9E+09,9E+09,9E+09]];
    CONST robtarget Target_6190:=[[84.528,89.711,0],[0.122788976,0.696364034,-0.696364034,0.122788976],[0, 0, 0, 0],[9E+09,9E+09,9E+09,9E+09,9E+09,9E+09]];
    CONST robtarget Target_6200:=[[106.352,127.511,0],[0.122788976,0.696364034,-0.696364034,0.122788976],[0, 0, 0, 0],[9E+09,9E+09,9E+09,9E+09,9E+09,9E+09]];
    CONST robtarget Target_6210:=[[193.648,127.511,0],[0.122788976,0.696364034,-0.696364034,0.122788976],[0, 0, 0, 0],[9E+09,9E+09,9E+09,9E+09,9E+09,9E+09]];
    CONST robtarget Target_6220:=[[215.471,89.711,0],[0.122788976,0.696364034,-0.696364034,0.122788976],[0, 0, 0, 0],[9E+09,9E+09,9E+09,9E+09,9E+09,9E+09]];
    CONST robtarget Target_6230:=[[174.081,89.711,0],[0.122788976,0.696364034,-0.696364034,0.122788976],[0, 0, 0, 0],[9E+09,9E+09,9E+09,9E+09,9E+09,9E+09]];
    CONST robtarget Target_6240:=[[150,127.511,0],[0.122788976,0.696364034,-0.696364034,0.122788976],[0, 0, 0, 0],[9E+09,9E+09,9E+09,9E+09,9E+09,9E+09]];
    CONST robtarget Target_6250:=[[130.498,169.333,0],[0.122788976,0.696364034,-0.696364034,0.122788976],[0, 0, 0, 0],[9E+09,9E+09,9E+09,9E+09,9E+09,9E+09]];
    CONST robtarget Target_6260:=[[150,203.111,0],[0.122788976,0.696364034,-0.696364034,0.122788976],[0, 0, 0, 0],[9E+09,9E+09,9E+09,9E+09,9E+09,9E+09]];
    CONST robtarget Target_6270:=[[169.502,169.333,0],[0.122788976,0.696364034,-0.696364034,0.122788976],[0, 0, 0, 0],[9E+09,9E+09,9E+09,9E+09,9E+09,9E+09]];
    CONST robtarget Target_6280:=[[150,127.511,0],[0.122788976,0.696364034,-0.696364034,0.122788976],[0, 0, 0, 0],[9E+09,9E+09,9E+09,9E+09,9E+09,9E+09]];
    CONST robtarget Target_6290:=[[125.919,89.711,0],[0.122788976,0.696364034,-0.696364034,0.122788976],[0, 0, 0, 0],[9E+09,9E+09,9E+09,9E+09,9E+09,9E+09]];
    CONST robtarget Target_6300:=[[84.528,89.711,0],[0.122788976,0.696364034,-0.696364034,0.122788976],[0, 0, 0, 0],[9E+09,9E+09,9E+09,9E+09,9E+09,9E+09]];
    CONST robtarget Target_6310:=[[84.528,89.711,20.7],[0.122788976,0.696364034,-0.696364034,0.122788976],[0, 0, 0, 0],[9E+09,9E+09,9E+09,9E+09,9E+09,9E+09]];
    CONST robtarget Target_6320:=[[71.457,55.472,20.7],[0.122788976,0.696364034,-0.696364034,0.122788976],[0, 0, 0, 0],[9E+09,9E+09,9E+09,9E+09,9E+09,9E+09]];
    CONST robtarget Target_6330:=[[71.457,55.472,0],[0.122788976,0.696364034,-0.696364034,0.122788976],[0, 0, 0, 0],[9E+09,9E+09,9E+09,9E+09,9E+09,9E+09]];
    CONST robtarget Target_6340:=[[71.457,76.472,0],[0.122788976,0.696364034,-0.696364034,0.122788976],[0, 0, 0, 0],[9E+09,9E+09,9E+09,9E+09,9E+09,9E+09]];
    CONST robtarget Target_6350:=[[75.269,76.472,0],[0.122788976,0.696364034,-0.696364034,0.122788976],[0, 0, 0, 0],[9E+09,9E+09,9E+09,9E+09,9E+09,9E+09]];
    CONST robtarget Target_6360:=[[80.51,64.78,0],[0.122788976,0.696364034,-0.696364034,0.122788976],[0, 0, 0, 0],[9E+09,9E+09,9E+09,9E+09,9E+09,9E+09]];
    CONST robtarget Target_6370:=[[85.582,76.472,0],[0.122788976,0.696364034,-0.696364034,0.122788976],[0, 0, 0, 0],[9E+09,9E+09,9E+09,9E+09,9E+09,9E+09]];
    CONST robtarget Target_6380:=[[89.462,76.472,0],[0.122788976,0.696364034,-0.696364034,0.122788976],[0, 0, 0, 0],[9E+09,9E+09,9E+09,9E+09,9E+09,9E+09]];
    CONST robtarget Target_6390:=[[89.462,55.472,0],[0.122788976,0.696364034,-0.696364034,0.122788976],[0, 0, 0, 0],[9E+09,9E+09,9E+09,9E+09,9E+09,9E+09]];
    CONST robtarget Target_6400:=[[89.462,55.472,20.7],[0.122788976,0.696364034,-0.696364034,0.122788976],[0, 0, 0, 0],[9E+09,9E+09,9E+09,9E+09,9E+09,9E+09]];
    CONST robtarget Target_6410:=[[92.899,55.472,20.7],[0.122788976,0.696364034,-0.696364034,0.122788976],[0, 0, 0, 0],[9E+09,9E+09,9E+09,9E+09,9E+09,9E+09]];
    CONST robtarget Target_6420:=[[92.899,55.472,0],[0.122788976,0.696364034,-0.696364034,0.122788976],[0, 0, 0, 0],[9E+09,9E+09,9E+09,9E+09,9E+09,9E+09]];
    CONST robtarget Target_6430:=[[101.034,55.472,0],[0.122788976,0.696364034,-0.696364034,0.122788976],[0, 0, 0, 0],[9E+09,9E+09,9E+09,9E+09,9E+09,9E+09]];
    CONST robtarget Target_6440:=[[96.967,55.472,0],[0.122788976,0.696364034,-0.696364034,0.122788976],[0, 0, 0, 0],[9E+09,9E+09,9E+09,9E+09,9E+09,9E+09]];
    CONST robtarget Target_6450:=[[96.967,76.472,0],[0.122788976,0.696364034,-0.696364034,0.122788976],[0, 0, 0, 0],[9E+09,9E+09,9E+09,9E+09,9E+09,9E+09]];
    CONST robtarget Target_6460:=[[92.899,76.472,0],[0.122788976,0.696364034,-0.696364034,0.122788976],[0, 0, 0, 0],[9E+09,9E+09,9E+09,9E+09,9E+09,9E+09]];
    CONST robtarget Target_6470:=[[101.034,76.472,0],[0.122788976,0.696364034,-0.696364034,0.122788976],[0, 0, 0, 0],[9E+09,9E+09,9E+09,9E+09,9E+09,9E+09]];
    CONST robtarget Target_6480:=[[101.034,76.472,20.7],[0.122788976,0.696364034,-0.696364034,0.122788976],[0, 0, 0, 0],[9E+09,9E+09,9E+09,9E+09,9E+09,9E+09]];
    CONST robtarget Target_6490:=[[102.344,76.472,20.7],[0.122788976,0.696364034,-0.696364034,0.122788976],[0, 0, 0, 0],[9E+09,9E+09,9E+09,9E+09,9E+09,9E+09]];
    CONST robtarget Target_6500:=[[102.344,76.472,0],[0.122788976,0.696364034,-0.696364034,0.122788976],[0, 0, 0, 0],[9E+09,9E+09,9E+09,9E+09,9E+09,9E+09]];
    CONST robtarget Target_6510:=[[119.226,76.472,0],[0.122788976,0.696364034,-0.696364034,0.122788976],[0, 0, 0, 0],[9E+09,9E+09,9E+09,9E+09,9E+09,9E+09]];
    CONST robtarget Target_6520:=[[110.785,76.472,0],[0.122788976,0.696364034,-0.696364034,0.122788976],[0, 0, 0, 0],[9E+09,9E+09,9E+09,9E+09,9E+09,9E+09]];
    CONST robtarget Target_6530:=[[110.785,55.472,0],[0.122788976,0.696364034,-0.696364034,0.122788976],[0, 0, 0, 0],[9E+09,9E+09,9E+09,9E+09,9E+09,9E+09]];
    CONST robtarget Target_6540:=[[110.785,55.472,20.7],[0.122788976,0.696364034,-0.696364034,0.122788976],[0, 0, 0, 0],[9E+09,9E+09,9E+09,9E+09,9E+09,9E+09]];
    CONST robtarget Target_6550:=[[120.315,56.731,20.7],[0.122788976,0.696364034,-0.696364034,0.122788976],[0, 0, 0, 0],[9E+09,9E+09,9E+09,9E+09,9E+09,9E+09]];
    CONST robtarget Target_6560:=[[120.315,56.731,0],[0.122788976,0.696364034,-0.696364034,0.122788976],[0, 0, 0, 0],[9E+09,9E+09,9E+09,9E+09,9E+09,9E+09]];
    CONST robtarget Target_6570:=[[123.327,55.574,0],[0.122788976,0.696364034,-0.696364034,0.122788976],[0, 0, 0, 0],[9E+09,9E+09,9E+09,9E+09,9E+09,9E+09]];
    CONST robtarget Target_6580:=[[127.207,55.097,0],[0.122788976,0.696364034,-0.696364034,0.122788976],[0, 0, 0, 0],[9E+09,9E+09,9E+09,9E+09,9E+09,9E+09]];
    CONST robtarget Target_6590:=[[130.407,55.591,0],[0.122788976,0.696364034,-0.696364034,0.122788976],[0, 0, 0, 0],[9E+09,9E+09,9E+09,9E+09,9E+09,9E+09]];
    CONST robtarget Target_6600:=[[132.687,57.003,0],[0.122788976,0.696364034,-0.696364034,0.122788976],[0, 0, 0, 0],[9E+09,9E+09,9E+09,9E+09,9E+09,9E+09]];
    CONST robtarget Target_6610:=[[134.091,59.028,0],[0.122788976,0.696364034,-0.696364034,0.122788976],[0, 0, 0, 0],[9E+09,9E+09,9E+09,9E+09,9E+09,9E+09]];
    CONST robtarget Target_6620:=[[134.593,61.462,0],[0.122788976,0.696364034,-0.696364034,0.122788976],[0, 0, 0, 0],[9E+09,9E+09,9E+09,9E+09,9E+09,9E+09]];
    CONST robtarget Target_6630:=[[133.589,64.755,0],[0.122788976,0.696364034,-0.696364034,0.122788976],[0, 0, 0, 0],[9E+09,9E+09,9E+09,9E+09,9E+09,9E+09]];
    CONST robtarget Target_6640:=[[130.424,66.754,0],[0.122788976,0.696364034,-0.696364034,0.122788976],[0, 0, 0, 0],[9E+09,9E+09,9E+09,9E+09,9E+09,9E+09]];
    CONST robtarget Target_6650:=[[128.288,67.316,0],[0.122788976,0.696364034,-0.696364034,0.122788976],[0, 0, 0, 0],[9E+09,9E+09,9E+09,9E+09,9E+09,9E+09]];
    CONST robtarget Target_6660:=[[126.118,67.861,0],[0.122788976,0.696364034,-0.696364034,0.122788976],[0, 0, 0, 0],[9E+09,9E+09,9E+09,9E+09,9E+09,9E+09]];
    CONST robtarget Target_6670:=[[124.084,69.009,0],[0.122788976,0.696364034,-0.696364034,0.122788976],[0, 0, 0, 0],[9E+09,9E+09,9E+09,9E+09,9E+09,9E+09]];
    CONST robtarget Target_6680:=[[123.378,71.128,0],[0.122788976,0.696364034,-0.696364034,0.122788976],[0, 0, 0, 0],[9E+09,9E+09,9E+09,9E+09,9E+09,9E+09]];
    CONST robtarget Target_6690:=[[124.578,73.519,0],[0.122788976,0.696364034,-0.696364034,0.122788976],[0, 0, 0, 0],[9E+09,9E+09,9E+09,9E+09,9E+09,9E+09]];
    CONST robtarget Target_6700:=[[127.718,74.429,0],[0.122788976,0.696364034,-0.696364034,0.122788976],[0, 0, 0, 0],[9E+09,9E+09,9E+09,9E+09,9E+09,9E+09]];
    CONST robtarget Target_6710:=[[131.002,73.749,0],[0.122788976,0.696364034,-0.696364034,0.122788976],[0, 0, 0, 0],[9E+09,9E+09,9E+09,9E+09,9E+09,9E+09]];
    CONST robtarget Target_6720:=[[133.572,72.149,0],[0.122788976,0.696364034,-0.696364034,0.122788976],[0, 0, 0, 0],[9E+09,9E+09,9E+09,9E+09,9E+09,9E+09]];
    CONST robtarget Target_6730:=[[133.572,72.149,20.7],[0.122788976,0.696364034,-0.696364034,0.122788976],[0, 0, 0, 0],[9E+09,9E+09,9E+09,9E+09,9E+09,9E+09]];
    CONST robtarget Target_6740:=[[137.18,76.472,20.7],[0.122788976,0.696364034,-0.696364034,0.122788976],[0, 0, 0, 0],[9E+09,9E+09,9E+09,9E+09,9E+09,9E+09]];
    CONST robtarget Target_6750:=[[137.18,76.472,0],[0.122788976,0.696364034,-0.696364034,0.122788976],[0, 0, 0, 0],[9E+09,9E+09,9E+09,9E+09,9E+09,9E+09]];
    CONST robtarget Target_6760:=[[137.18,69.92,0],[0.122788976,0.696364034,-0.696364034,0.122788976],[0, 0, 0, 0],[9E+09,9E+09,9E+09,9E+09,9E+09,9E+09]];
    CONST robtarget Target_6770:=[[137.18,63.368,0],[0.122788976,0.696364034,-0.696364034,0.122788976],[0, 0, 0, 0],[9E+09,9E+09,9E+09,9E+09,9E+09,9E+09]];
    CONST robtarget Target_6780:=[[137.631,59.59,0],[0.122788976,0.696364034,-0.696364034,0.122788976],[0, 0, 0, 0],[9E+09,9E+09,9E+09,9E+09,9E+09,9E+09]];
    CONST robtarget Target_6790:=[[139.188,56.969,0],[0.122788976,0.696364034,-0.696364034,0.122788976],[0, 0, 0, 0],[9E+09,9E+09,9E+09,9E+09,9E+09,9E+09]];
    CONST robtarget Target_6800:=[[141.536,55.514,0],[0.122788976,0.696364034,-0.696364034,0.122788976],[0, 0, 0, 0],[9E+09,9E+09,9E+09,9E+09,9E+09,9E+09]];
    CONST robtarget Target_6810:=[[144.77,55.029,0],[0.122788976,0.696364034,-0.696364034,0.122788976],[0, 0, 0, 0],[9E+09,9E+09,9E+09,9E+09,9E+09,9E+09]];
    CONST robtarget Target_6820:=[[148.037,55.506,0],[0.122788976,0.696364034,-0.696364034,0.122788976],[0, 0, 0, 0],[9E+09,9E+09,9E+09,9E+09,9E+09,9E+09]];
    CONST robtarget Target_6830:=[[150.368,56.969,0],[0.122788976,0.696364034,-0.696364034,0.122788976],[0, 0, 0, 0],[9E+09,9E+09,9E+09,9E+09,9E+09,9E+09]];
    CONST robtarget Target_6840:=[[151.934,59.607,0],[0.122788976,0.696364034,-0.696364034,0.122788976],[0, 0, 0, 0],[9E+09,9E+09,9E+09,9E+09,9E+09,9E+09]];
    CONST robtarget Target_6850:=[[152.377,63.368,0],[0.122788976,0.696364034,-0.696364034,0.122788976],[0, 0, 0, 0],[9E+09,9E+09,9E+09,9E+09,9E+09,9E+09]];
    CONST robtarget Target_6860:=[[152.377,69.92,0],[0.122788976,0.696364034,-0.696364034,0.122788976],[0, 0, 0, 0],[9E+09,9E+09,9E+09,9E+09,9E+09,9E+09]];
    CONST robtarget Target_6870:=[[152.377,76.472,0],[0.122788976,0.696364034,-0.696364034,0.122788976],[0, 0, 0, 0],[9E+09,9E+09,9E+09,9E+09,9E+09,9E+09]];
    CONST robtarget Target_6880:=[[152.377,76.472,20.7],[0.122788976,0.696364034,-0.696364034,0.122788976],[0, 0, 0, 0],[9E+09,9E+09,9E+09,9E+09,9E+09,9E+09]];
    CONST robtarget Target_6890:=[[156.376,76.472,20.7],[0.122788976,0.696364034,-0.696364034,0.122788976],[0, 0, 0, 0],[9E+09,9E+09,9E+09,9E+09,9E+09,9E+09]];
    CONST robtarget Target_6900:=[[156.376,76.472,0],[0.122788976,0.696364034,-0.696364034,0.122788976],[0, 0, 0, 0],[9E+09,9E+09,9E+09,9E+09,9E+09,9E+09]];
    CONST robtarget Target_6910:=[[156.376,55.472,0],[0.122788976,0.696364034,-0.696364034,0.122788976],[0, 0, 0, 0],[9E+09,9E+09,9E+09,9E+09,9E+09,9E+09]];
    CONST robtarget Target_6920:=[[162.4,55.472,0],[0.122788976,0.696364034,-0.696364034,0.122788976],[0, 0, 0, 0],[9E+09,9E+09,9E+09,9E+09,9E+09,9E+09]];
    CONST robtarget Target_6930:=[[165.897,55.863,0],[0.122788976,0.696364034,-0.696364034,0.122788976],[0, 0, 0, 0],[9E+09,9E+09,9E+09,9E+09,9E+09,9E+09]];
    CONST robtarget Target_6940:=[[168.441,57.173,0],[0.122788976,0.696364034,-0.696364034,0.122788976],[0, 0, 0, 0],[9E+09,9E+09,9E+09,9E+09,9E+09,9E+09]];
    CONST robtarget Target_6950:=[[170.024,59.156,0],[0.122788976,0.696364034,-0.696364034,0.122788976],[0, 0, 0, 0],[9E+09,9E+09,9E+09,9E+09,9E+09,9E+09]];
    CONST robtarget Target_6960:=[[170.62,61.921,0],[0.122788976,0.696364034,-0.696364034,0.122788976],[0, 0, 0, 0],[9E+09,9E+09,9E+09,9E+09,9E+09,9E+09]];
    CONST robtarget Target_6970:=[[169.59,65.282,0],[0.122788976,0.696364034,-0.696364034,0.122788976],[0, 0, 0, 0],[9E+09,9E+09,9E+09,9E+09,9E+09,9E+09]];
    CONST robtarget Target_6980:=[[166.689,67.248,0],[0.122788976,0.696364034,-0.696364034,0.122788976],[0, 0, 0, 0],[9E+09,9E+09,9E+09,9E+09,9E+09,9E+09]];
    CONST robtarget Target_6990:=[[156.376,65.972,0],[0.122788976,0.696364034,-0.696364034,0.122788976],[0, 0, 0, 0],[9E+09,9E+09,9E+09,9E+09,9E+09,9E+09]];
    CONST robtarget Target_7000:=[[166.689,67.248,0],[0.122788976,0.696364034,-0.696364034,0.122788976],[0, 0, 0, 0],[9E+09,9E+09,9E+09,9E+09,9E+09,9E+09]];
    CONST robtarget Target_7010:=[[168.85,69.086,0],[0.122788976,0.696364034,-0.696364034,0.122788976],[0, 0, 0, 0],[9E+09,9E+09,9E+09,9E+09,9E+09,9E+09]];
    CONST robtarget Target_7020:=[[169.633,71.741,0],[0.122788976,0.696364034,-0.696364034,0.122788976],[0, 0, 0, 0],[9E+09,9E+09,9E+09,9E+09,9E+09,9E+09]];
    CONST robtarget Target_7030:=[[169.114,74.047,0],[0.122788976,0.696364034,-0.696364034,0.122788976],[0, 0, 0, 0],[9E+09,9E+09,9E+09,9E+09,9E+09,9E+09]];
    CONST robtarget Target_7040:=[[167.454,75.621,0],[0.122788976,0.696364034,-0.696364034,0.122788976],[0, 0, 0, 0],[9E+09,9E+09,9E+09,9E+09,9E+09,9E+09]];
    CONST robtarget Target_7050:=[[161.941,76.472,0],[0.122788976,0.696364034,-0.696364034,0.122788976],[0, 0, 0, 0],[9E+09,9E+09,9E+09,9E+09,9E+09,9E+09]];
    CONST robtarget Target_7060:=[[156.376,76.472,0],[0.122788976,0.696364034,-0.696364034,0.122788976],[0, 0, 0, 0],[9E+09,9E+09,9E+09,9E+09,9E+09,9E+09]];
    CONST robtarget Target_7070:=[[156.376,76.472,20.7],[0.122788976,0.696364034,-0.696364034,0.122788976],[0, 0, 0, 0],[9E+09,9E+09,9E+09,9E+09,9E+09,9E+09]];
    CONST robtarget Target_7080:=[[172.577,76.472,20.7],[0.122788976,0.696364034,-0.696364034,0.122788976],[0, 0, 0, 0],[9E+09,9E+09,9E+09,9E+09,9E+09,9E+09]];
    CONST robtarget Target_7090:=[[172.577,76.472,0],[0.122788976,0.696364034,-0.696364034,0.122788976],[0, 0, 0, 0],[9E+09,9E+09,9E+09,9E+09,9E+09,9E+09]];
    CONST robtarget Target_7100:=[[180.711,76.472,0],[0.122788976,0.696364034,-0.696364034,0.122788976],[0, 0, 0, 0],[9E+09,9E+09,9E+09,9E+09,9E+09,9E+09]];
    CONST robtarget Target_7110:=[[176.644,76.472,0],[0.122788976,0.696364034,-0.696364034,0.122788976],[0, 0, 0, 0],[9E+09,9E+09,9E+09,9E+09,9E+09,9E+09]];
    CONST robtarget Target_7120:=[[176.644,55.472,0],[0.122788976,0.696364034,-0.696364034,0.122788976],[0, 0, 0, 0],[9E+09,9E+09,9E+09,9E+09,9E+09,9E+09]];
    CONST robtarget Target_7130:=[[172.577,55.472,0],[0.122788976,0.696364034,-0.696364034,0.122788976],[0, 0, 0, 0],[9E+09,9E+09,9E+09,9E+09,9E+09,9E+09]];
    CONST robtarget Target_7140:=[[180.711,55.472,0],[0.122788976,0.696364034,-0.696364034,0.122788976],[0, 0, 0, 0],[9E+09,9E+09,9E+09,9E+09,9E+09,9E+09]];
    CONST robtarget Target_7150:=[[180.711,55.472,20.7],[0.122788976,0.696364034,-0.696364034,0.122788976],[0, 0, 0, 0],[9E+09,9E+09,9E+09,9E+09,9E+09,9E+09]];
    CONST robtarget Target_7160:=[[183.128,56.731,20.7],[0.122788976,0.696364034,-0.696364034,0.122788976],[0, 0, 0, 0],[9E+09,9E+09,9E+09,9E+09,9E+09,9E+09]];
    CONST robtarget Target_7170:=[[183.128,56.731,0],[0.122788976,0.696364034,-0.696364034,0.122788976],[0, 0, 0, 0],[9E+09,9E+09,9E+09,9E+09,9E+09,9E+09]];
    CONST robtarget Target_7180:=[[190.02,55.097,0],[0.122788976,0.696364034,-0.696364034,0.122788976],[0, 0, 0, 0],[9E+09,9E+09,9E+09,9E+09,9E+09,9E+09]];
    CONST robtarget Target_7190:=[[193.219,55.591,0],[0.122788976,0.696364034,-0.696364034,0.122788976],[0, 0, 0, 0],[9E+09,9E+09,9E+09,9E+09,9E+09,9E+09]];
    CONST robtarget Target_7200:=[[195.5,57.003,0],[0.122788976,0.696364034,-0.696364034,0.122788976],[0, 0, 0, 0],[9E+09,9E+09,9E+09,9E+09,9E+09,9E+09]];
    CONST robtarget Target_7210:=[[196.904,59.028,0],[0.122788976,0.696364034,-0.696364034,0.122788976],[0, 0, 0, 0],[9E+09,9E+09,9E+09,9E+09,9E+09,9E+09]];
    CONST robtarget Target_7220:=[[197.406,61.462,0],[0.122788976,0.696364034,-0.696364034,0.122788976],[0, 0, 0, 0],[9E+09,9E+09,9E+09,9E+09,9E+09,9E+09]];
    CONST robtarget Target_7230:=[[196.402,64.755,0],[0.122788976,0.696364034,-0.696364034,0.122788976],[0, 0, 0, 0],[9E+09,9E+09,9E+09,9E+09,9E+09,9E+09]];
    CONST robtarget Target_7240:=[[193.236,66.754,0],[0.122788976,0.696364034,-0.696364034,0.122788976],[0, 0, 0, 0],[9E+09,9E+09,9E+09,9E+09,9E+09,9E+09]];
    CONST robtarget Target_7250:=[[191.101,67.316,0],[0.122788976,0.696364034,-0.696364034,0.122788976],[0, 0, 0, 0],[9E+09,9E+09,9E+09,9E+09,9E+09,9E+09]];
    CONST robtarget Target_7260:=[[188.931,67.861,0],[0.122788976,0.696364034,-0.696364034,0.122788976],[0, 0, 0, 0],[9E+09,9E+09,9E+09,9E+09,9E+09,9E+09]];
    CONST robtarget Target_7270:=[[186.897,69.009,0],[0.122788976,0.696364034,-0.696364034,0.122788976],[0, 0, 0, 0],[9E+09,9E+09,9E+09,9E+09,9E+09,9E+09]];
    CONST robtarget Target_7280:=[[186.191,71.128,0],[0.122788976,0.696364034,-0.696364034,0.122788976],[0, 0, 0, 0],[9E+09,9E+09,9E+09,9E+09,9E+09,9E+09]];
    CONST robtarget Target_7290:=[[187.391,73.519,0],[0.122788976,0.696364034,-0.696364034,0.122788976],[0, 0, 0, 0],[9E+09,9E+09,9E+09,9E+09,9E+09,9E+09]];
    CONST robtarget Target_7300:=[[190.531,74.429,0],[0.122788976,0.696364034,-0.696364034,0.122788976],[0, 0, 0, 0],[9E+09,9E+09,9E+09,9E+09,9E+09,9E+09]];
    CONST robtarget Target_7310:=[[193.815,73.749,0],[0.122788976,0.696364034,-0.696364034,0.122788976],[0, 0, 0, 0],[9E+09,9E+09,9E+09,9E+09,9E+09,9E+09]];
    CONST robtarget Target_7320:=[[196.385,72.149,0],[0.122788976,0.696364034,-0.696364034,0.122788976],[0, 0, 0, 0],[9E+09,9E+09,9E+09,9E+09,9E+09,9E+09]];
    CONST robtarget Target_7330:=[[196.385,72.149,20.7],[0.122788976,0.696364034,-0.696364034,0.122788976],[0, 0, 0, 0],[9E+09,9E+09,9E+09,9E+09,9E+09,9E+09]];
    CONST robtarget Target_7340:=[[200.248,76.472,20.7],[0.122788976,0.696364034,-0.696364034,0.122788976],[0, 0, 0, 0],[9E+09,9E+09,9E+09,9E+09,9E+09,9E+09]];
    CONST robtarget Target_7350:=[[200.248,76.472,0],[0.122788976,0.696364034,-0.696364034,0.122788976],[0, 0, 0, 0],[9E+09,9E+09,9E+09,9E+09,9E+09,9E+09]];
    CONST robtarget Target_7360:=[[200.248,55.472,0],[0.122788976,0.696364034,-0.696364034,0.122788976],[0, 0, 0, 0],[9E+09,9E+09,9E+09,9E+09,9E+09,9E+09]];
    CONST robtarget Target_7370:=[[200.248,65.972,0],[0.122788976,0.696364034,-0.696364034,0.122788976],[0, 0, 0, 0],[9E+09,9E+09,9E+09,9E+09,9E+09,9E+09]];
    CONST robtarget Target_7380:=[[215.496,65.972,0],[0.122788976,0.696364034,-0.696364034,0.122788976],[0, 0, 0, 0],[9E+09,9E+09,9E+09,9E+09,9E+09,9E+09]];
    CONST robtarget Target_7390:=[[215.496,55.472,0],[0.122788976,0.696364034,-0.696364034,0.122788976],[0, 0, 0, 0],[9E+09,9E+09,9E+09,9E+09,9E+09,9E+09]];
    CONST robtarget Target_7400:=[[215.496,76.472,0],[0.122788976,0.696364034,-0.696364034,0.122788976],[0, 0, 0, 0],[9E+09,9E+09,9E+09,9E+09,9E+09,9E+09]];
    CONST robtarget Target_7410:=[[215.496,76.472,20.7],[0.122788976,0.696364034,-0.696364034,0.122788976],[0, 0, 0, 0],[9E+09,9E+09,9E+09,9E+09,9E+09,9E+09]];
    CONST robtarget Target_7420:=[[218.933,76.472,20.7],[0.122788976,0.696364034,-0.696364034,0.122788976],[0, 0, 0, 0],[9E+09,9E+09,9E+09,9E+09,9E+09,9E+09]];
    CONST robtarget Target_7430:=[[218.933,76.472,0],[0.122788976,0.696364034,-0.696364034,0.122788976],[0, 0, 0, 0],[9E+09,9E+09,9E+09,9E+09,9E+09,9E+09]];
    CONST robtarget Target_7440:=[[227.068,76.472,0],[0.122788976,0.696364034,-0.696364034,0.122788976],[0, 0, 0, 0],[9E+09,9E+09,9E+09,9E+09,9E+09,9E+09]];
    CONST robtarget Target_7450:=[[223.001,76.472,0],[0.122788976,0.696364034,-0.696364034,0.122788976],[0, 0, 0, 0],[9E+09,9E+09,9E+09,9E+09,9E+09,9E+09]];
    CONST robtarget Target_7460:=[[223.001,55.472,0],[0.122788976,0.696364034,-0.696364034,0.122788976],[0, 0, 0, 0],[9E+09,9E+09,9E+09,9E+09,9E+09,9E+09]];
    CONST robtarget Target_7470:=[[218.933,55.472,0],[0.122788976,0.696364034,-0.696364034,0.122788976],[0, 0, 0, 0],[9E+09,9E+09,9E+09,9E+09,9E+09,9E+09]];
    CONST robtarget Target_7480:=[[227.068,55.472,0],[0.122788976,0.696364034,-0.696364034,0.122788976],[0, 0, 0, 0],[9E+09,9E+09,9E+09,9E+09,9E+09,9E+09]];
    CONST robtarget Target_7490:=[[227.068,55.472,20.7],[0.122788976,0.696364034,-0.696364034,0.122788976],[0, 0, 0, 0],[9E+09,9E+09,9E+09,9E+09,9E+09,9E+09]];
    CONST robtarget Target_7500:=[[93.988,20.896,20.7],[0.122788976,0.696364034,-0.696364034,0.122788976],[0, 0, 0, 0],[9E+09,9E+09,9E+09,9E+09,9E+09,9E+09]];
    CONST robtarget Target_7510:=[[93.988,20.896,0],[0.122788976,0.696364034,-0.696364034,0.122788976],[0, 0, 0, 0],[9E+09,9E+09,9E+09,9E+09,9E+09,9E+09]];
    CONST robtarget Target_7520:=[[93.988,41.896,0],[0.122788976,0.696364034,-0.696364034,0.122788976],[0, 0, 0, 0],[9E+09,9E+09,9E+09,9E+09,9E+09,9E+09]];
    CONST robtarget Target_7530:=[[97.8,41.896,0],[0.122788976,0.696364034,-0.696364034,0.122788976],[0, 0, 0, 0],[9E+09,9E+09,9E+09,9E+09,9E+09,9E+09]];
    CONST robtarget Target_7540:=[[103.042,30.204,0],[0.122788976,0.696364034,-0.696364034,0.122788976],[0, 0, 0, 0],[9E+09,9E+09,9E+09,9E+09,9E+09,9E+09]];
    CONST robtarget Target_7550:=[[108.113,41.896,0],[0.122788976,0.696364034,-0.696364034,0.122788976],[0, 0, 0, 0],[9E+09,9E+09,9E+09,9E+09,9E+09,9E+09]];
    CONST robtarget Target_7560:=[[111.993,41.896,0],[0.122788976,0.696364034,-0.696364034,0.122788976],[0, 0, 0, 0],[9E+09,9E+09,9E+09,9E+09,9E+09,9E+09]];
    CONST robtarget Target_7570:=[[111.993,20.896,0],[0.122788976,0.696364034,-0.696364034,0.122788976],[0, 0, 0, 0],[9E+09,9E+09,9E+09,9E+09,9E+09,9E+09]];
    CONST robtarget Target_7580:=[[111.993,20.896,20.7],[0.122788976,0.696364034,-0.696364034,0.122788976],[0, 0, 0, 0],[9E+09,9E+09,9E+09,9E+09,9E+09,9E+09]];
    CONST robtarget Target_7590:=[[115.056,31.396,0],[0.122788976,0.696364034,-0.696364034,0.122788976],[0, 0, 0, 0],[9E+09,9E+09,9E+09,9E+09,9E+09,9E+09]];
    CONST robtarget Target_7600:=[[115.703,26.758,0],[0.122788976,0.696364034,-0.696364034,0.122788976],[0, 0, 0, 0],[9E+09,9E+09,9E+09,9E+09,9E+09,9E+09]];
    CONST robtarget Target_7610:=[[117.558,23.312,0],[0.122788976,0.696364034,-0.696364034,0.122788976],[0, 0, 0, 0],[9E+09,9E+09,9E+09,9E+09,9E+09,9E+09]];
    CONST robtarget Target_7620:=[[120.502,21.176,0],[0.122788976,0.696364034,-0.696364034,0.122788976],[0, 0, 0, 0],[9E+09,9E+09,9E+09,9E+09,9E+09,9E+09]];
    CONST robtarget Target_7630:=[[124.331,20.453,0],[0.122788976,0.696364034,-0.696364034,0.122788976],[0, 0, 0, 0],[9E+09,9E+09,9E+09,9E+09,9E+09,9E+09]];
    CONST robtarget Target_7640:=[[128.101,21.151,0],[0.122788976,0.696364034,-0.696364034,0.122788976],[0, 0, 0, 0],[9E+09,9E+09,9E+09,9E+09,9E+09,9E+09]];
    CONST robtarget Target_7650:=[[131.104,23.312,0],[0.122788976,0.696364034,-0.696364034,0.122788976],[0, 0, 0, 0],[9E+09,9E+09,9E+09,9E+09,9E+09,9E+09]];
    CONST robtarget Target_7660:=[[132.976,26.775,0],[0.122788976,0.696364034,-0.696364034,0.122788976],[0, 0, 0, 0],[9E+09,9E+09,9E+09,9E+09,9E+09,9E+09]];
    CONST robtarget Target_7670:=[[133.623,31.396,0],[0.122788976,0.696364034,-0.696364034,0.122788976],[0, 0, 0, 0],[9E+09,9E+09,9E+09,9E+09,9E+09,9E+09]];
    CONST robtarget Target_7680:=[[132.959,36.058,0],[0.122788976,0.696364034,-0.696364034,0.122788976],[0, 0, 0, 0],[9E+09,9E+09,9E+09,9E+09,9E+09,9E+09]];
    CONST robtarget Target_7690:=[[131.104,39.496,0],[0.122788976,0.696364034,-0.696364034,0.122788976],[0, 0, 0, 0],[9E+09,9E+09,9E+09,9E+09,9E+09,9E+09]];
    CONST robtarget Target_7700:=[[128.194,41.589,0],[0.122788976,0.696364034,-0.696364034,0.122788976],[0, 0, 0, 0],[9E+09,9E+09,9E+09,9E+09,9E+09,9E+09]];
    CONST robtarget Target_7710:=[[124.331,42.338,0],[0.122788976,0.696364034,-0.696364034,0.122788976],[0, 0, 0, 0],[9E+09,9E+09,9E+09,9E+09,9E+09,9E+09]];
    CONST robtarget Target_7720:=[[120.511,41.615,0],[0.122788976,0.696364034,-0.696364034,0.122788976],[0, 0, 0, 0],[9E+09,9E+09,9E+09,9E+09,9E+09,9E+09]];
    CONST robtarget Target_7730:=[[117.575,39.496,0],[0.122788976,0.696364034,-0.696364034,0.122788976],[0, 0, 0, 0],[9E+09,9E+09,9E+09,9E+09,9E+09,9E+09]];
    CONST robtarget Target_7740:=[[115.712,36.041,0],[0.122788976,0.696364034,-0.696364034,0.122788976],[0, 0, 0, 0],[9E+09,9E+09,9E+09,9E+09,9E+09,9E+09]];
    CONST robtarget Target_7750:=[[115.056,31.396,0],[0.122788976,0.696364034,-0.696364034,0.122788976],[0, 0, 0, 0],[9E+09,9E+09,9E+09,9E+09,9E+09,9E+09]];
    CONST robtarget Target_7760:=[[115.056,31.396,20.7],[0.122788976,0.696364034,-0.696364034,0.122788976],[0, 0, 0, 0],[9E+09,9E+09,9E+09,9E+09,9E+09,9E+09]];
    CONST robtarget Target_7770:=[[134.542,41.896,20.7],[0.122788976,0.696364034,-0.696364034,0.122788976],[0, 0, 0, 0],[9E+09,9E+09,9E+09,9E+09,9E+09,9E+09]];
    CONST robtarget Target_7780:=[[134.542,41.896,0],[0.122788976,0.696364034,-0.696364034,0.122788976],[0, 0, 0, 0],[9E+09,9E+09,9E+09,9E+09,9E+09,9E+09]];
    CONST robtarget Target_7790:=[[151.424,41.896,0],[0.122788976,0.696364034,-0.696364034,0.122788976],[0, 0, 0, 0],[9E+09,9E+09,9E+09,9E+09,9E+09,9E+09]];
    CONST robtarget Target_7800:=[[142.983,41.896,0],[0.122788976,0.696364034,-0.696364034,0.122788976],[0, 0, 0, 0],[9E+09,9E+09,9E+09,9E+09,9E+09,9E+09]];
    CONST robtarget Target_7810:=[[142.983,20.896,0],[0.122788976,0.696364034,-0.696364034,0.122788976],[0, 0, 0, 0],[9E+09,9E+09,9E+09,9E+09,9E+09,9E+09]];
    CONST robtarget Target_7820:=[[142.983,20.896,20.7],[0.122788976,0.696364034,-0.696364034,0.122788976],[0, 0, 0, 0],[9E+09,9E+09,9E+09,9E+09,9E+09,9E+09]];
    CONST robtarget Target_7830:=[[152.36,31.396,20.7],[0.122788976,0.696364034,-0.696364034,0.122788976],[0, 0, 0, 0],[9E+09,9E+09,9E+09,9E+09,9E+09,9E+09]];
    CONST robtarget Target_7840:=[[152.36,31.396,0],[0.122788976,0.696364034,-0.696364034,0.122788976],[0, 0, 0, 0],[9E+09,9E+09,9E+09,9E+09,9E+09,9E+09]];
    CONST robtarget Target_7850:=[[153.006,26.758,0],[0.122788976,0.696364034,-0.696364034,0.122788976],[0, 0, 0, 0],[9E+09,9E+09,9E+09,9E+09,9E+09,9E+09]];
    CONST robtarget Target_7860:=[[154.861,23.312,0],[0.122788976,0.696364034,-0.696364034,0.122788976],[0, 0, 0, 0],[9E+09,9E+09,9E+09,9E+09,9E+09,9E+09]];
    CONST robtarget Target_7870:=[[157.805,21.176,0],[0.122788976,0.696364034,-0.696364034,0.122788976],[0, 0, 0, 0],[9E+09,9E+09,9E+09,9E+09,9E+09,9E+09]];
    CONST robtarget Target_7880:=[[161.634,20.453,0],[0.122788976,0.696364034,-0.696364034,0.122788976],[0, 0, 0, 0],[9E+09,9E+09,9E+09,9E+09,9E+09,9E+09]];
    CONST robtarget Target_7890:=[[165.404,21.151,0],[0.122788976,0.696364034,-0.696364034,0.122788976],[0, 0, 0, 0],[9E+09,9E+09,9E+09,9E+09,9E+09,9E+09]];
    CONST robtarget Target_7900:=[[168.407,23.312,0],[0.122788976,0.696364034,-0.696364034,0.122788976],[0, 0, 0, 0],[9E+09,9E+09,9E+09,9E+09,9E+09,9E+09]];
    CONST robtarget Target_7910:=[[170.279,26.775,0],[0.122788976,0.696364034,-0.696364034,0.122788976],[0, 0, 0, 0],[9E+09,9E+09,9E+09,9E+09,9E+09,9E+09]];
    CONST robtarget Target_7920:=[[170.926,31.396,0],[0.122788976,0.696364034,-0.696364034,0.122788976],[0, 0, 0, 0],[9E+09,9E+09,9E+09,9E+09,9E+09,9E+09]];
    CONST robtarget Target_7930:=[[170.262,36.058,0],[0.122788976,0.696364034,-0.696364034,0.122788976],[0, 0, 0, 0],[9E+09,9E+09,9E+09,9E+09,9E+09,9E+09]];
    CONST robtarget Target_7940:=[[168.407,39.496,0],[0.122788976,0.696364034,-0.696364034,0.122788976],[0, 0, 0, 0],[9E+09,9E+09,9E+09,9E+09,9E+09,9E+09]];
    CONST robtarget Target_7950:=[[165.497,41.589,0],[0.122788976,0.696364034,-0.696364034,0.122788976],[0, 0, 0, 0],[9E+09,9E+09,9E+09,9E+09,9E+09,9E+09]];
    CONST robtarget Target_7960:=[[161.634,42.338,0],[0.122788976,0.696364034,-0.696364034,0.122788976],[0, 0, 0, 0],[9E+09,9E+09,9E+09,9E+09,9E+09,9E+09]];
    CONST robtarget Target_7970:=[[157.814,41.615,0],[0.122788976,0.696364034,-0.696364034,0.122788976],[0, 0, 0, 0],[9E+09,9E+09,9E+09,9E+09,9E+09,9E+09]];
    CONST robtarget Target_7980:=[[154.878,39.496,0],[0.122788976,0.696364034,-0.696364034,0.122788976],[0, 0, 0, 0],[9E+09,9E+09,9E+09,9E+09,9E+09,9E+09]];
    CONST robtarget Target_7990:=[[153.015,36.041,0],[0.122788976,0.696364034,-0.696364034,0.122788976],[0, 0, 0, 0],[9E+09,9E+09,9E+09,9E+09,9E+09,9E+09]];
    CONST robtarget Target_8000:=[[152.36,31.396,0],[0.122788976,0.696364034,-0.696364034,0.122788976],[0, 0, 0, 0],[9E+09,9E+09,9E+09,9E+09,9E+09,9E+09]];
    CONST robtarget Target_8010:=[[152.36,31.396,20.7],[0.122788976,0.696364034,-0.696364034,0.122788976],[0, 0, 0, 0],[9E+09,9E+09,9E+09,9E+09,9E+09,9E+09]];
    CONST robtarget Target_8020:=[[173.989,41.896,20.7],[0.122788976,0.696364034,-0.696364034,0.122788976],[0, 0, 0, 0],[9E+09,9E+09,9E+09,9E+09,9E+09,9E+09]];
    CONST robtarget Target_8030:=[[173.989,41.896,0],[0.122788976,0.696364034,-0.696364034,0.122788976],[0, 0, 0, 0],[9E+09,9E+09,9E+09,9E+09,9E+09,9E+09]];
    CONST robtarget Target_8040:=[[173.989,20.896,0],[0.122788976,0.696364034,-0.696364034,0.122788976],[0, 0, 0, 0],[9E+09,9E+09,9E+09,9E+09,9E+09,9E+09]];
    CONST robtarget Target_8050:=[[173.989,41.896,0],[0.122788976,0.696364034,-0.696364034,0.122788976],[0, 0, 0, 0],[9E+09,9E+09,9E+09,9E+09,9E+09,9E+09]];
    CONST robtarget Target_8060:=[[179.401,41.896,0],[0.122788976,0.696364034,-0.696364034,0.122788976],[0, 0, 0, 0],[9E+09,9E+09,9E+09,9E+09,9E+09,9E+09]];
    CONST robtarget Target_8070:=[[182.422,41.7,0],[0.122788976,0.696364034,-0.696364034,0.122788976],[0, 0, 0, 0],[9E+09,9E+09,9E+09,9E+09,9E+09,9E+09]];
    CONST robtarget Target_8080:=[[184.745,40.789,0],[0.122788976,0.696364034,-0.696364034,0.122788976],[0, 0, 0, 0],[9E+09,9E+09,9E+09,9E+09,9E+09,9E+09]];
    CONST robtarget Target_8090:=[[186.489,38.96,0],[0.122788976,0.696364034,-0.696364034,0.122788976],[0, 0, 0, 0],[9E+09,9E+09,9E+09,9E+09,9E+09,9E+09]];
    CONST robtarget Target_8100:=[[187.127,36.195,0],[0.122788976,0.696364034,-0.696364034,0.122788976],[0, 0, 0, 0],[9E+09,9E+09,9E+09,9E+09,9E+09,9E+09]];
    CONST robtarget Target_8110:=[[185.953,32.34,0],[0.122788976,0.696364034,-0.696364034,0.122788976],[0, 0, 0, 0],[9E+09,9E+09,9E+09,9E+09,9E+09,9E+09]];
    CONST robtarget Target_8120:=[[182.77,30.034,0],[0.122788976,0.696364034,-0.696364034,0.122788976],[0, 0, 0, 0],[9E+09,9E+09,9E+09,9E+09,9E+09,9E+09]];
    CONST robtarget Target_8130:=[[176.78,29.251,0],[0.122788976,0.696364034,-0.696364034,0.122788976],[0, 0, 0, 0],[9E+09,9E+09,9E+09,9E+09,9E+09,9E+09]];
    CONST robtarget Target_8140:=[[182.77,30.034,0],[0.122788976,0.696364034,-0.696364034,0.122788976],[0, 0, 0, 0],[9E+09,9E+09,9E+09,9E+09,9E+09,9E+09]];
    CONST robtarget Target_8150:=[[190.241,20.896,0],[0.122788976,0.696364034,-0.696364034,0.122788976],[0, 0, 0, 0],[9E+09,9E+09,9E+09,9E+09,9E+09,9E+09]];
    CONST robtarget Target_8160:=[[190.241,20.896,20.7],[0.122788976,0.696364034,-0.696364034,0.122788976],[0, 0, 0, 0],[9E+09,9E+09,9E+09,9E+09,9E+09,9E+09]];
    CONST robtarget Target_8170:=[[190.871,22.155,20.7],[0.122788976,0.696364034,-0.696364034,0.122788976],[0, 0, 0, 0],[9E+09,9E+09,9E+09,9E+09,9E+09,9E+09]];
    CONST robtarget Target_8180:=[[190.871,22.155,0],[0.122788976,0.696364034,-0.696364034,0.122788976],[0, 0, 0, 0],[9E+09,9E+09,9E+09,9E+09,9E+09,9E+09]];
    CONST robtarget Target_8190:=[[197.763,20.521,0],[0.122788976,0.696364034,-0.696364034,0.122788976],[0, 0, 0, 0],[9E+09,9E+09,9E+09,9E+09,9E+09,9E+09]];
    CONST robtarget Target_8200:=[[200.962,21.015,0],[0.122788976,0.696364034,-0.696364034,0.122788976],[0, 0, 0, 0],[9E+09,9E+09,9E+09,9E+09,9E+09,9E+09]];
    CONST robtarget Target_8210:=[[203.243,22.427,0],[0.122788976,0.696364034,-0.696364034,0.122788976],[0, 0, 0, 0],[9E+09,9E+09,9E+09,9E+09,9E+09,9E+09]];
    CONST robtarget Target_8220:=[[204.647,24.452,0],[0.122788976,0.696364034,-0.696364034,0.122788976],[0, 0, 0, 0],[9E+09,9E+09,9E+09,9E+09,9E+09,9E+09]];
    CONST robtarget Target_8230:=[[205.149,26.886,0],[0.122788976,0.696364034,-0.696364034,0.122788976],[0, 0, 0, 0],[9E+09,9E+09,9E+09,9E+09,9E+09,9E+09]];
    CONST robtarget Target_8240:=[[204.145,30.179,0],[0.122788976,0.696364034,-0.696364034,0.122788976],[0, 0, 0, 0],[9E+09,9E+09,9E+09,9E+09,9E+09,9E+09]];
    CONST robtarget Target_8250:=[[200.98,32.178,0],[0.122788976,0.696364034,-0.696364034,0.122788976],[0, 0, 0, 0],[9E+09,9E+09,9E+09,9E+09,9E+09,9E+09]];
    CONST robtarget Target_8260:=[[198.844,32.74,0],[0.122788976,0.696364034,-0.696364034,0.122788976],[0, 0, 0, 0],[9E+09,9E+09,9E+09,9E+09,9E+09,9E+09]];
    CONST robtarget Target_8270:=[[196.674,33.285,0],[0.122788976,0.696364034,-0.696364034,0.122788976],[0, 0, 0, 0],[9E+09,9E+09,9E+09,9E+09,9E+09,9E+09]];
    CONST robtarget Target_8280:=[[194.64,34.433,0],[0.122788976,0.696364034,-0.696364034,0.122788976],[0, 0, 0, 0],[9E+09,9E+09,9E+09,9E+09,9E+09,9E+09]];
    CONST robtarget Target_8290:=[[193.934,36.552,0],[0.122788976,0.696364034,-0.696364034,0.122788976],[0, 0, 0, 0],[9E+09,9E+09,9E+09,9E+09,9E+09,9E+09]];
    CONST robtarget Target_8300:=[[195.134,38.943,0],[0.122788976,0.696364034,-0.696364034,0.122788976],[0, 0, 0, 0],[9E+09,9E+09,9E+09,9E+09,9E+09,9E+09]];
    CONST robtarget Target_8310:=[[198.274,39.853,0],[0.122788976,0.696364034,-0.696364034,0.122788976],[0, 0, 0, 0],[9E+09,9E+09,9E+09,9E+09,9E+09,9E+09]];
    CONST robtarget Target_8320:=[[201.558,39.173,0],[0.122788976,0.696364034,-0.696364034,0.122788976],[0, 0, 0, 0],[9E+09,9E+09,9E+09,9E+09,9E+09,9E+09]];
    CONST robtarget Target_8330:=[[204.128,37.573,0],[0.122788976,0.696364034,-0.696364034,0.122788976],[0, 0, 0, 0],[9E+09,9E+09,9E+09,9E+09,9E+09,9E+09]];
    CONST robtarget Maintenance:=[[-536.273831699,-715.042774725,569.87661133],[0.198438475,0.442588128,0.101109453,-0.868628113],[0, 0, 0, 0],[9E+09,9E+09,9E+09,9E+09,9E+09,9E+09]];

    PROC Path_10()
        MoveL Target_4030,v300,z1,TCP\WObj:=Workobject_5;
        MoveL Target_4040,v300,z1,TCP\WObj:=Workobject_5;
        MoveL Target_4050,v300,z1,TCP\WObj:=Workobject_5;
        MoveL Target_4060,v300,z1,TCP\WObj:=Workobject_5;
        MoveL Target_4070,v300,z1,TCP\WObj:=Workobject_5;
        MoveL Target_4080,v300,z1,TCP\WObj:=Workobject_5;
        MoveL Target_4090,v300,z1,TCP\WObj:=Workobject_5;
        MoveL Target_4100,v300,z1,TCP\WObj:=Workobject_5;
        MoveL Target_4110,v300,z1,TCP\WObj:=Workobject_5;
        MoveL Target_4120,v300,z1,TCP\WObj:=Workobject_5;
        MoveL Target_4130,v300,z1,TCP\WObj:=Workobject_5;
        MoveL Target_4140,v300,z1,TCP\WObj:=Workobject_5;
        MoveL Target_4150,v300,z1,TCP\WObj:=Workobject_5;
        MoveL Target_4160,v300,z1,TCP\WObj:=Workobject_5;
        MoveL Target_4170,v300,z1,TCP\WObj:=Workobject_5;
        MoveL Target_4180,v300,z1,TCP\WObj:=Workobject_5;
        MoveL Target_4190,v300,z1,TCP\WObj:=Workobject_5;
        MoveL Target_4200,v300,z1,TCP\WObj:=Workobject_5;
        MoveL Target_4210,v300,z1,TCP\WObj:=Workobject_5;
        MoveL Target_4220,v300,z1,TCP\WObj:=Workobject_5;
        MoveL Target_4230,v300,z1,TCP\WObj:=Workobject_5;
        MoveL Target_4240,v300,z1,TCP\WObj:=Workobject_5;
        MoveL Target_4250,v300,z1,TCP\WObj:=Workobject_5;
        MoveL Target_4260,v300,z1,TCP\WObj:=Workobject_5;
        MoveL Target_4270,v300,z1,TCP\WObj:=Workobject_5;
        MoveL Target_4280,v300,z1,TCP\WObj:=Workobject_5;
        MoveL Target_4290,v300,z1,TCP\WObj:=Workobject_5;
        MoveL Target_4300,v300,z1,TCP\WObj:=Workobject_5;
        MoveL Target_4310,v300,z1,TCP\WObj:=Workobject_5;
        MoveL Target_4320,v300,z1,TCP\WObj:=Workobject_5;
        MoveL Target_4330,v300,z1,TCP\WObj:=Workobject_5;
        MoveL Target_4340,v300,z1,TCP\WObj:=Workobject_5;
        MoveL Target_4350,v300,z1,TCP\WObj:=Workobject_5;
        MoveL Target_4360,v300,z1,TCP\WObj:=Workobject_5;
        MoveL Target_4370,v300,z1,TCP\WObj:=Workobject_5;
        MoveL Target_4380,v300,z1,TCP\WObj:=Workobject_5;
        MoveL Target_4390,v300,z1,TCP\WObj:=Workobject_5;
        MoveL Target_4400,v300,z1,TCP\WObj:=Workobject_5;
        MoveL Target_4410,v300,z1,TCP\WObj:=Workobject_5;
        MoveL Target_4420,v300,z1,TCP\WObj:=Workobject_5;
        MoveL Target_4430,v300,z1,TCP\WObj:=Workobject_5;
        MoveL Target_4440,v300,z1,TCP\WObj:=Workobject_5;
        MoveL Target_4450,v300,z1,TCP\WObj:=Workobject_5;
        MoveL Target_4460,v300,z1,TCP\WObj:=Workobject_5;
        MoveL Target_4470,v300,z1,TCP\WObj:=Workobject_5;
        MoveL Target_4480,v300,z1,TCP\WObj:=Workobject_5;
        MoveL Target_4490,v300,z1,TCP\WObj:=Workobject_5;
        MoveL Target_4500,v300,z1,TCP\WObj:=Workobject_5;
        MoveL Target_4510,v300,z1,TCP\WObj:=Workobject_5;
        MoveL Target_4520,v300,z1,TCP\WObj:=Workobject_5;
        MoveL Target_4530,v300,z1,TCP\WObj:=Workobject_5;
        MoveL Target_4540,v300,z1,TCP\WObj:=Workobject_5;
        MoveL Target_4550,v300,z1,TCP\WObj:=Workobject_5;
        MoveL Target_4560,v300,z1,TCP\WObj:=Workobject_5;
        MoveL Target_4570,v300,z1,TCP\WObj:=Workobject_5;
        MoveL Target_4580,v300,z1,TCP\WObj:=Workobject_5;
        MoveL Target_4590,v300,z1,TCP\WObj:=Workobject_5;
        MoveL Target_4600,v300,z1,TCP\WObj:=Workobject_5;
        MoveL Target_4610,v300,z1,TCP\WObj:=Workobject_5;
        MoveL Target_4620,v300,z1,TCP\WObj:=Workobject_5;
        MoveL Target_4630,v300,z1,TCP\WObj:=Workobject_5;
        MoveL Target_4640,v300,z1,TCP\WObj:=Workobject_5;
        MoveL Target_4650,v300,z1,TCP\WObj:=Workobject_5;
        MoveL Target_4660,v300,z1,TCP\WObj:=Workobject_5;
        MoveL Target_4670,v300,z1,TCP\WObj:=Workobject_5;
        MoveL Target_4680,v300,z1,TCP\WObj:=Workobject_5;
        MoveL Target_4690,v300,z1,TCP\WObj:=Workobject_5;
        MoveL Target_4700,v300,z1,TCP\WObj:=Workobject_5;
        MoveL Target_4710,v300,z1,TCP\WObj:=Workobject_5;
        MoveL Target_4720,v300,z1,TCP\WObj:=Workobject_5;
        MoveL Target_4730,v300,z1,TCP\WObj:=Workobject_5;
        MoveL Target_4740,v300,z1,TCP\WObj:=Workobject_5;
        MoveL Target_4750,v300,z1,TCP\WObj:=Workobject_5;
        MoveL Target_4760,v300,z1,TCP\WObj:=Workobject_5;
        MoveL Target_4770,v300,z1,TCP\WObj:=Workobject_5;
        MoveL Target_4780,v300,z1,TCP\WObj:=Workobject_5;
        MoveL Target_4790,v300,z1,TCP\WObj:=Workobject_5;
        MoveL Target_4800,v300,z1,TCP\WObj:=Workobject_5;
        MoveL Target_4810,v300,z1,TCP\WObj:=Workobject_5;
        MoveL Target_4820,v300,z1,TCP\WObj:=Workobject_5;
        MoveL Target_4830,v300,z1,TCP\WObj:=Workobject_5;
        MoveL Target_4840,v300,z1,TCP\WObj:=Workobject_5;
        MoveL Target_4850,v300,z1,TCP\WObj:=Workobject_5;
        MoveL Target_4860,v300,z1,TCP\WObj:=Workobject_5;
        MoveL Target_4870,v300,z1,TCP\WObj:=Workobject_5;
        MoveL Target_4880,v300,z1,TCP\WObj:=Workobject_5;
        MoveL Target_4890,v300,z1,TCP\WObj:=Workobject_5;
        MoveL Target_4900,v300,z1,TCP\WObj:=Workobject_5;
        MoveL Target_4910,v300,z1,TCP\WObj:=Workobject_5;
        MoveL Target_4920,v300,z1,TCP\WObj:=Workobject_5;
        MoveL Target_4930,v300,z1,TCP\WObj:=Workobject_5;
        MoveL Target_4940,v300,z1,TCP\WObj:=Workobject_5;
        MoveL Target_4950,v300,z1,TCP\WObj:=Workobject_5;
        MoveL Target_4960,v300,z1,TCP\WObj:=Workobject_5;
        MoveL Target_4970,v300,z1,TCP\WObj:=Workobject_5;
        MoveL Target_4980,v300,z1,TCP\WObj:=Workobject_5;
        MoveL Target_4990,v300,z1,TCP\WObj:=Workobject_5;
        MoveL Target_5000,v300,z1,TCP\WObj:=Workobject_5;
        MoveL Target_5010,v300,z1,TCP\WObj:=Workobject_5;
        MoveL Target_5020,v300,z1,TCP\WObj:=Workobject_5;
        MoveL Target_5030,v300,z1,TCP\WObj:=Workobject_5;
        MoveL Target_5040,v300,z1,TCP\WObj:=Workobject_5;
        MoveL Target_5050,v300,z1,TCP\WObj:=Workobject_5;
        MoveL Target_5060,v300,z1,TCP\WObj:=Workobject_5;
        MoveL Target_5070,v300,z1,TCP\WObj:=Workobject_5;
        MoveL Target_5080,v300,z1,TCP\WObj:=Workobject_5;
        MoveL Target_5090,v300,z1,TCP\WObj:=Workobject_5;
        MoveL Target_5100,v300,z1,TCP\WObj:=Workobject_5;
        MoveL Target_5110,v300,z1,TCP\WObj:=Workobject_5;
        MoveL Target_5120,v300,z1,TCP\WObj:=Workobject_5;
        MoveL Target_5130,v300,z1,TCP\WObj:=Workobject_5;
        MoveL Target_5140,v300,z1,TCP\WObj:=Workobject_5;
        MoveL Target_5150,v300,z1,TCP\WObj:=Workobject_5;
        MoveL Target_5160,v300,z1,TCP\WObj:=Workobject_5;
        MoveL Target_5170,v300,z1,TCP\WObj:=Workobject_5;
        MoveL Target_5180,v300,z1,TCP\WObj:=Workobject_5;
        MoveL Target_5190,v300,z1,TCP\WObj:=Workobject_5;
        MoveL Target_5200,v300,z1,TCP\WObj:=Workobject_5;
        MoveL Target_5210,v300,z1,TCP\WObj:=Workobject_5;
        MoveL Target_5220,v300,z1,TCP\WObj:=Workobject_5;
        MoveL Target_5230,v300,z1,TCP\WObj:=Workobject_5;
        MoveL Target_5240,v300,z1,TCP\WObj:=Workobject_5;
        MoveL Target_5250,v300,z1,TCP\WObj:=Workobject_5;
        MoveL Target_5260,v300,z1,TCP\WObj:=Workobject_5;
        MoveL Target_5270,v300,z1,TCP\WObj:=Workobject_5;
        MoveL Target_5280,v300,z1,TCP\WObj:=Workobject_5;
        MoveL Target_5290,v300,z1,TCP\WObj:=Workobject_5;
        MoveL Target_5300,v300,z1,TCP\WObj:=Workobject_5;
        MoveL Target_5310,v300,z1,TCP\WObj:=Workobject_5;
        MoveL Target_5320,v300,z1,TCP\WObj:=Workobject_5;
        MoveL Target_5330,v300,z1,TCP\WObj:=Workobject_5;
        MoveL Target_5340,v300,z1,TCP\WObj:=Workobject_5;
        MoveL Target_5350,v300,z1,TCP\WObj:=Workobject_5;
        MoveL Target_5360,v300,z1,TCP\WObj:=Workobject_5;
        MoveL Target_5370,v300,z1,TCP\WObj:=Workobject_5;
        MoveL Target_5380,v300,z1,TCP\WObj:=Workobject_5;
        MoveL Target_5390,v300,z1,TCP\WObj:=Workobject_5;
        MoveL Target_5400,v300,z1,TCP\WObj:=Workobject_5;
        MoveL Target_5410,v300,z1,TCP\WObj:=Workobject_5;
        MoveL Target_5420,v300,z1,TCP\WObj:=Workobject_5;
        MoveL Target_5430,v300,z1,TCP\WObj:=Workobject_5;
        MoveL Target_5440,v300,z1,TCP\WObj:=Workobject_5;
        MoveL Target_5450,v300,z1,TCP\WObj:=Workobject_5;
        MoveL Target_5460,v300,z1,TCP\WObj:=Workobject_5;
        MoveL Target_5470,v300,z1,TCP\WObj:=Workobject_5;
        MoveL Target_5480,v300,z1,TCP\WObj:=Workobject_5;
        MoveL Target_5490,v300,z1,TCP\WObj:=Workobject_5;
        MoveL Target_5500,v300,z1,TCP\WObj:=Workobject_5;
        MoveL Target_5510,v300,z1,TCP\WObj:=Workobject_5;
        MoveL Target_5520,v300,z1,TCP\WObj:=Workobject_5;
        MoveL Target_5530,v300,z1,TCP\WObj:=Workobject_5;
        MoveL Target_5540,v300,z1,TCP\WObj:=Workobject_5;
        MoveL Target_5550,v300,z1,TCP\WObj:=Workobject_5;
        MoveL Target_5560,v300,z1,TCP\WObj:=Workobject_5;
        MoveL Target_5570,v300,z1,TCP\WObj:=Workobject_5;
        MoveL Target_5580,v300,z1,TCP\WObj:=Workobject_5;
        MoveL Target_5590,v300,z1,TCP\WObj:=Workobject_5;
        MoveL Target_5600,v300,z1,TCP\WObj:=Workobject_5;
        MoveL Target_5610,v300,z1,TCP\WObj:=Workobject_5;
        MoveL Target_5620,v300,z1,TCP\WObj:=Workobject_5;
        MoveL Target_5630,v300,z1,TCP\WObj:=Workobject_5;
        MoveL Target_5640,v300,z1,TCP\WObj:=Workobject_5;
        MoveL Target_5650,v300,z1,TCP\WObj:=Workobject_5;
        MoveL Target_5660,v300,z1,TCP\WObj:=Workobject_5;
        MoveL Target_5670,v300,z1,TCP\WObj:=Workobject_5;
        MoveL Target_5680,v300,z1,TCP\WObj:=Workobject_5;
        MoveL Target_5690,v300,z1,TCP\WObj:=Workobject_5;
        MoveL Target_5700,v300,z1,TCP\WObj:=Workobject_5;
        MoveL Target_5710,v300,z1,TCP\WObj:=Workobject_5;
        MoveL Target_5720,v300,z1,TCP\WObj:=Workobject_5;
        MoveL Target_5730,v300,z1,TCP\WObj:=Workobject_5;
        MoveL Target_5740,v300,z1,TCP\WObj:=Workobject_5;
        MoveL Target_5750,v300,z1,TCP\WObj:=Workobject_5;
        MoveL Target_5760,v300,z1,TCP\WObj:=Workobject_5;
        MoveL Target_5770,v300,z1,TCP\WObj:=Workobject_5;
        MoveL Target_5780,v300,z1,TCP\WObj:=Workobject_5;
        MoveL Target_5790,v300,z1,TCP\WObj:=Workobject_5;
        MoveL Target_5800,v300,z1,TCP\WObj:=Workobject_5;
        MoveL Target_5810,v300,z1,TCP\WObj:=Workobject_5;
        MoveL Target_5820,v300,z1,TCP\WObj:=Workobject_5;
        MoveL Target_5830,v300,z1,TCP\WObj:=Workobject_5;
        MoveL Target_5840,v300,z1,TCP\WObj:=Workobject_5;
        MoveL Target_5850,v300,z1,TCP\WObj:=Workobject_5;
        MoveL Target_5860,v300,z1,TCP\WObj:=Workobject_5;
        MoveL Target_5870,v300,z1,TCP\WObj:=Workobject_5;
        MoveL Target_5880,v300,z1,TCP\WObj:=Workobject_5;
        MoveL Target_5890,v300,z1,TCP\WObj:=Workobject_5;
        MoveL Target_5900,v300,z1,TCP\WObj:=Workobject_5;
        MoveL Target_5910,v300,z1,TCP\WObj:=Workobject_5;
        MoveL Target_5920,v300,z1,TCP\WObj:=Workobject_5;
        MoveL Target_5930,v300,z1,TCP\WObj:=Workobject_5;
        MoveL Target_5940,v300,z1,TCP\WObj:=Workobject_5;
        MoveL Target_5950,v300,z1,TCP\WObj:=Workobject_5;
        MoveL Target_5960,v300,z1,TCP\WObj:=Workobject_5;
        MoveL Target_5970,v300,z1,TCP\WObj:=Workobject_5;
        MoveL Target_5980,v300,z1,TCP\WObj:=Workobject_5;
        MoveL Target_5990,v300,z1,TCP\WObj:=Workobject_5;
        MoveL Target_6000,v300,z1,TCP\WObj:=Workobject_5;
        MoveL Target_6010,v300,z1,TCP\WObj:=Workobject_5;
        MoveL Target_6020,v300,z1,TCP\WObj:=Workobject_5;
        MoveL Target_6030,v300,z1,TCP\WObj:=Workobject_5;
        MoveL Target_6040,v300,z1,TCP\WObj:=Workobject_5;
        MoveL Target_6050,v300,z1,TCP\WObj:=Workobject_5;
        MoveL Target_6060,v300,z1,TCP\WObj:=Workobject_5;
        MoveL Target_6070,v300,z1,TCP\WObj:=Workobject_5;
        MoveL Target_6080,v300,z1,TCP\WObj:=Workobject_5;
        MoveL Target_6090,v300,z1,TCP\WObj:=Workobject_5;
        MoveL Target_6100,v300,z1,TCP\WObj:=Workobject_5;
        MoveL Target_6110,v300,z1,TCP\WObj:=Workobject_5;
        MoveL Target_6120,v300,z1,TCP\WObj:=Workobject_5;
        MoveL Target_6130,v300,z1,TCP\WObj:=Workobject_5;
        MoveL Target_6140,v300,z1,TCP\WObj:=Workobject_5;
        MoveL Target_6150,v300,z1,TCP\WObj:=Workobject_5;
        MoveL Target_6160,v300,z1,TCP\WObj:=Workobject_5;
        MoveL Target_6170,v300,z1,TCP\WObj:=Workobject_5;
        MoveL Target_6180,v300,z1,TCP\WObj:=Workobject_5;
        MoveJ HOME,v300,z1,TCP\WObj:=Workobject_5;
    ENDPROC
    PROC main()
        WaitDI DI_01,1;
        SetDO DO_01,1;
        Path_10;
        Path_20;
        WaitDI DI_02,1;
        Path_30;
        Reset DO_01;
    ENDPROC
    PROC Path_20()
        MoveL Target_6190,v300,z1,TCP\WObj:=Workobject_6;
        MoveL Target_6200,v300,z1,TCP\WObj:=Workobject_6;
        MoveL Target_6210,v300,z1,TCP\WObj:=Workobject_6;
        MoveL Target_6220,v300,z1,TCP\WObj:=Workobject_6;
        MoveL Target_6230,v300,z1,TCP\WObj:=Workobject_6;
        MoveL Target_6240,v300,z1,TCP\WObj:=Workobject_6;
        MoveL Target_6250,v300,z1,TCP\WObj:=Workobject_6;
        MoveL Target_6260,v300,z1,TCP\WObj:=Workobject_6;
        MoveL Target_6270,v300,z1,TCP\WObj:=Workobject_6;
        MoveL Target_6280,v300,z1,TCP\WObj:=Workobject_6;
        MoveL Target_6290,v300,z1,TCP\WObj:=Workobject_6;
        MoveL Target_6300,v300,z1,TCP\WObj:=Workobject_6;
        MoveL Target_6310,v300,z1,TCP\WObj:=Workobject_6;
        MoveL Target_6320,v300,z1,TCP\WObj:=Workobject_6;
        MoveL Target_6330,v300,z1,TCP\WObj:=Workobject_6;
        MoveL Target_6340,v300,z1,TCP\WObj:=Workobject_6;
        MoveL Target_6350,v300,z1,TCP\WObj:=Workobject_6;
        MoveL Target_6360,v300,z1,TCP\WObj:=Workobject_6;
        MoveL Target_6370,v300,z1,TCP\WObj:=Workobject_6;
        MoveL Target_6380,v300,z1,TCP\WObj:=Workobject_6;
        MoveL Target_6390,v300,z1,TCP\WObj:=Workobject_6;
        MoveL Target_6400,v300,z1,TCP\WObj:=Workobject_6;
        MoveL Target_6410,v300,z1,TCP\WObj:=Workobject_6;
        MoveL Target_6420,v300,z1,TCP\WObj:=Workobject_6;
        MoveL Target_6430,v300,z1,TCP\WObj:=Workobject_6;
        MoveL Target_6440,v300,z1,TCP\WObj:=Workobject_6;
        MoveL Target_6450,v300,z1,TCP\WObj:=Workobject_6;
        MoveL Target_6460,v300,z1,TCP\WObj:=Workobject_6;
        MoveL Target_6470,v300,z1,TCP\WObj:=Workobject_6;
        MoveL Target_6480,v300,z1,TCP\WObj:=Workobject_6;
        MoveL Target_6490,v300,z1,TCP\WObj:=Workobject_6;
        MoveL Target_6500,v300,z1,TCP\WObj:=Workobject_6;
        MoveL Target_6510,v300,z1,TCP\WObj:=Workobject_6;
        MoveL Target_6520,v300,z1,TCP\WObj:=Workobject_6;
        MoveL Target_6530,v300,z1,TCP\WObj:=Workobject_6;
        MoveL Target_6540,v300,z1,TCP\WObj:=Workobject_6;
        MoveL Target_6550,v300,z1,TCP\WObj:=Workobject_6;
        MoveL Target_6560,v300,z1,TCP\WObj:=Workobject_6;
        MoveL Target_6570,v300,z1,TCP\WObj:=Workobject_6;
        MoveL Target_6580,v300,z1,TCP\WObj:=Workobject_6;
        MoveL Target_6590,v300,z1,TCP\WObj:=Workobject_6;
        MoveL Target_6600,v300,z1,TCP\WObj:=Workobject_6;
        MoveL Target_6610,v300,z1,TCP\WObj:=Workobject_6;
        MoveL Target_6620,v300,z1,TCP\WObj:=Workobject_6;
        MoveL Target_6630,v300,z1,TCP\WObj:=Workobject_6;
        MoveL Target_6640,v300,z1,TCP\WObj:=Workobject_6;
        MoveL Target_6650,v300,z1,TCP\WObj:=Workobject_6;
        MoveL Target_6660,v300,z1,TCP\WObj:=Workobject_6;
        MoveL Target_6670,v300,z1,TCP\WObj:=Workobject_6;
        MoveL Target_6680,v300,z1,TCP\WObj:=Workobject_6;
        MoveL Target_6690,v300,z1,TCP\WObj:=Workobject_6;
        MoveL Target_6700,v300,z1,TCP\WObj:=Workobject_6;
        MoveL Target_6710,v300,z1,TCP\WObj:=Workobject_6;
        MoveL Target_6720,v300,z1,TCP\WObj:=Workobject_6;
        MoveL Target_6730,v300,z1,TCP\WObj:=Workobject_6;
        MoveL Target_6740,v300,z1,TCP\WObj:=Workobject_6;
        MoveL Target_6750,v300,z1,TCP\WObj:=Workobject_6;
        MoveL Target_6760,v300,z1,TCP\WObj:=Workobject_6;
        MoveL Target_6770,v300,z1,TCP\WObj:=Workobject_6;
        MoveL Target_6780,v300,z1,TCP\WObj:=Workobject_6;
        MoveL Target_6790,v300,z1,TCP\WObj:=Workobject_6;
        MoveL Target_6800,v300,z1,TCP\WObj:=Workobject_6;
        MoveL Target_6810,v300,z1,TCP\WObj:=Workobject_6;
        MoveL Target_6820,v300,z1,TCP\WObj:=Workobject_6;
        MoveL Target_6830,v300,z1,TCP\WObj:=Workobject_6;
        MoveL Target_6840,v300,z1,TCP\WObj:=Workobject_6;
        MoveL Target_6850,v300,z1,TCP\WObj:=Workobject_6;
        MoveL Target_6860,v300,z1,TCP\WObj:=Workobject_6;
        MoveL Target_6870,v300,z1,TCP\WObj:=Workobject_6;
        MoveL Target_6880,v300,z1,TCP\WObj:=Workobject_6;
        MoveL Target_6890,v300,z1,TCP\WObj:=Workobject_6;
        MoveL Target_6900,v300,z1,TCP\WObj:=Workobject_6;
        MoveL Target_6910,v300,z1,TCP\WObj:=Workobject_6;
        MoveL Target_6920,v300,z1,TCP\WObj:=Workobject_6;
        MoveL Target_6930,v300,z1,TCP\WObj:=Workobject_6;
        MoveL Target_6940,v300,z1,TCP\WObj:=Workobject_6;
        MoveL Target_6950,v300,z1,TCP\WObj:=Workobject_6;
        MoveL Target_6960,v300,z1,TCP\WObj:=Workobject_6;
        MoveL Target_6970,v300,z1,TCP\WObj:=Workobject_6;
        MoveL Target_6980,v300,z1,TCP\WObj:=Workobject_6;
        MoveL Target_6990,v300,z1,TCP\WObj:=Workobject_6;
        MoveL Target_7000,v300,z1,TCP\WObj:=Workobject_6;
        MoveL Target_7010,v300,z1,TCP\WObj:=Workobject_6;
        MoveL Target_7020,v300,z1,TCP\WObj:=Workobject_6;
        MoveL Target_7030,v300,z1,TCP\WObj:=Workobject_6;
        MoveL Target_7040,v300,z1,TCP\WObj:=Workobject_6;
        MoveL Target_7050,v300,z1,TCP\WObj:=Workobject_6;
        MoveL Target_7060,v300,z1,TCP\WObj:=Workobject_6;
        MoveL Target_7070,v300,z1,TCP\WObj:=Workobject_6;
        MoveL Target_7080,v300,z1,TCP\WObj:=Workobject_6;
        MoveL Target_7090,v300,z1,TCP\WObj:=Workobject_6;
        MoveL Target_7100,v300,z1,TCP\WObj:=Workobject_6;
        MoveL Target_7110,v300,z1,TCP\WObj:=Workobject_6;
        MoveL Target_7120,v300,z1,TCP\WObj:=Workobject_6;
        MoveL Target_7130,v300,z1,TCP\WObj:=Workobject_6;
        MoveL Target_7140,v300,z1,TCP\WObj:=Workobject_6;
        MoveL Target_7150,v300,z1,TCP\WObj:=Workobject_6;
        MoveL Target_7160,v300,z1,TCP\WObj:=Workobject_6;
        MoveL Target_7170,v300,z1,TCP\WObj:=Workobject_6;
        MoveL Target_7180,v300,z1,TCP\WObj:=Workobject_6;
        MoveL Target_7190,v300,z1,TCP\WObj:=Workobject_6;
        MoveL Target_7200,v300,z1,TCP\WObj:=Workobject_6;
        MoveL Target_7210,v300,z1,TCP\WObj:=Workobject_6;
        MoveL Target_7220,v300,z1,TCP\WObj:=Workobject_6;
        MoveL Target_7230,v300,z1,TCP\WObj:=Workobject_6;
        MoveL Target_7240,v300,z1,TCP\WObj:=Workobject_6;
        MoveL Target_7250,v300,z1,TCP\WObj:=Workobject_6;
        MoveL Target_7260,v300,z1,TCP\WObj:=Workobject_6;
        MoveL Target_7270,v300,z1,TCP\WObj:=Workobject_6;
        MoveL Target_7280,v300,z1,TCP\WObj:=Workobject_6;
        MoveL Target_7290,v300,z1,TCP\WObj:=Workobject_6;
        MoveL Target_7300,v300,z1,TCP\WObj:=Workobject_6;
        MoveL Target_7310,v300,z1,TCP\WObj:=Workobject_6;
        MoveL Target_7320,v300,z1,TCP\WObj:=Workobject_6;
        MoveL Target_7330,v300,z1,TCP\WObj:=Workobject_6;
        MoveL Target_7340,v300,z1,TCP\WObj:=Workobject_6;
        MoveL Target_7350,v300,z1,TCP\WObj:=Workobject_6;
        MoveL Target_7360,v300,z1,TCP\WObj:=Workobject_6;
        MoveL Target_7370,v300,z1,TCP\WObj:=Workobject_6;
        MoveL Target_7380,v300,z1,TCP\WObj:=Workobject_6;
        MoveL Target_7390,v300,z1,TCP\WObj:=Workobject_6;
        MoveL Target_7400,v300,z1,TCP\WObj:=Workobject_6;
        MoveL Target_7410,v300,z1,TCP\WObj:=Workobject_6;
        MoveL Target_7420,v300,z1,TCP\WObj:=Workobject_6;
        MoveL Target_7430,v300,z1,TCP\WObj:=Workobject_6;
        MoveL Target_7440,v300,z1,TCP\WObj:=Workobject_6;
        MoveL Target_7450,v300,z1,TCP\WObj:=Workobject_6;
        MoveL Target_7460,v300,z1,TCP\WObj:=Workobject_6;
        MoveL Target_7470,v300,z1,TCP\WObj:=Workobject_6;
        MoveL Target_7480,v300,z1,TCP\WObj:=Workobject_6;
        MoveL Target_7490,v300,z1,TCP\WObj:=Workobject_6;
        MoveL Target_7500,v300,z1,TCP\WObj:=Workobject_6;
        MoveL Target_7510,v300,z1,TCP\WObj:=Workobject_6;
        MoveL Target_7520,v300,z1,TCP\WObj:=Workobject_6;
        MoveL Target_7530,v300,z1,TCP\WObj:=Workobject_6;
        MoveL Target_7540,v300,z1,TCP\WObj:=Workobject_6;
        MoveL Target_7550,v300,z1,TCP\WObj:=Workobject_6;
        MoveL Target_7560,v300,z1,TCP\WObj:=Workobject_6;
        MoveL Target_7570,v300,z1,TCP\WObj:=Workobject_6;
        MoveL Target_7580,v300,z1,TCP\WObj:=Workobject_6;
        MoveL Target_7590,v300,z1,TCP\WObj:=Workobject_6;
        MoveL Target_7600,v300,z1,TCP\WObj:=Workobject_6;
        MoveL Target_7610,v300,z1,TCP\WObj:=Workobject_6;
        MoveL Target_7620,v300,z1,TCP\WObj:=Workobject_6;
        MoveL Target_7630,v300,z1,TCP\WObj:=Workobject_6;
        MoveL Target_7640,v300,z1,TCP\WObj:=Workobject_6;
        MoveL Target_7650,v300,z1,TCP\WObj:=Workobject_6;
        MoveL Target_7660,v300,z1,TCP\WObj:=Workobject_6;
        MoveL Target_7670,v300,z1,TCP\WObj:=Workobject_6;
        MoveL Target_7680,v300,z1,TCP\WObj:=Workobject_6;
        MoveL Target_7690,v300,z1,TCP\WObj:=Workobject_6;
        MoveL Target_7700,v300,z1,TCP\WObj:=Workobject_6;
        MoveL Target_7710,v300,z1,TCP\WObj:=Workobject_6;
        MoveL Target_7720,v300,z1,TCP\WObj:=Workobject_6;
        MoveL Target_7730,v300,z1,TCP\WObj:=Workobject_6;
        MoveL Target_7740,v300,z1,TCP\WObj:=Workobject_6;
        MoveL Target_7750,v300,z1,TCP\WObj:=Workobject_6;
        MoveL Target_7760,v300,z1,TCP\WObj:=Workobject_6;
        MoveL Target_7770,v300,z1,TCP\WObj:=Workobject_6;
        MoveL Target_7780,v300,z1,TCP\WObj:=Workobject_6;
        MoveL Target_7790,v300,z1,TCP\WObj:=Workobject_6;
        MoveL Target_7800,v300,z1,TCP\WObj:=Workobject_6;
        MoveL Target_7810,v300,z1,TCP\WObj:=Workobject_6;
        MoveL Target_7820,v300,z1,TCP\WObj:=Workobject_6;
        MoveL Target_7830,v300,z1,TCP\WObj:=Workobject_6;
        MoveL Target_7840,v300,z1,TCP\WObj:=Workobject_6;
        MoveL Target_7850,v300,z1,TCP\WObj:=Workobject_6;
        MoveL Target_7860,v300,z1,TCP\WObj:=Workobject_6;
        MoveL Target_7870,v300,z1,TCP\WObj:=Workobject_6;
        MoveL Target_7880,v300,z1,TCP\WObj:=Workobject_6;
        MoveL Target_7890,v300,z1,TCP\WObj:=Workobject_6;
        MoveL Target_7900,v300,z1,TCP\WObj:=Workobject_6;
        MoveL Target_7910,v300,z1,TCP\WObj:=Workobject_6;
        MoveL Target_7920,v300,z1,TCP\WObj:=Workobject_6;
        MoveL Target_7930,v300,z1,TCP\WObj:=Workobject_6;
        MoveL Target_7940,v300,z1,TCP\WObj:=Workobject_6;
        MoveL Target_7950,v300,z1,TCP\WObj:=Workobject_6;
        MoveL Target_7960,v300,z1,TCP\WObj:=Workobject_6;
        MoveL Target_7970,v300,z1,TCP\WObj:=Workobject_6;
        MoveL Target_7980,v300,z1,TCP\WObj:=Workobject_6;
        MoveL Target_7990,v300,z1,TCP\WObj:=Workobject_6;
        MoveL Target_8000,v300,z1,TCP\WObj:=Workobject_6;
        MoveL Target_8010,v300,z1,TCP\WObj:=Workobject_6;
        MoveL Target_8020,v300,z1,TCP\WObj:=Workobject_6;
        MoveL Target_8030,v300,z1,TCP\WObj:=Workobject_6;
        MoveL Target_8040,v300,z1,TCP\WObj:=Workobject_6;
        MoveL Target_8050,v300,z1,TCP\WObj:=Workobject_6;
        MoveL Target_8060,v300,z1,TCP\WObj:=Workobject_6;
        MoveL Target_8070,v300,z1,TCP\WObj:=Workobject_6;
        MoveL Target_8080,v300,z1,TCP\WObj:=Workobject_6;
        MoveL Target_8090,v300,z1,TCP\WObj:=Workobject_6;
        MoveL Target_8100,v300,z1,TCP\WObj:=Workobject_6;
        MoveL Target_8110,v300,z1,TCP\WObj:=Workobject_6;
        MoveL Target_8120,v300,z1,TCP\WObj:=Workobject_6;
        MoveL Target_8130,v300,z1,TCP\WObj:=Workobject_6;
        MoveL Target_8140,v300,z1,TCP\WObj:=Workobject_6;
        MoveL Target_8150,v300,z1,TCP\WObj:=Workobject_6;
        MoveL Target_8160,v300,z1,TCP\WObj:=Workobject_6;
        MoveL Target_8170,v300,z1,TCP\WObj:=Workobject_6;
        MoveL Target_8180,v300,z1,TCP\WObj:=Workobject_6;
        MoveL Target_8190,v300,z1,TCP\WObj:=Workobject_6;
        MoveL Target_8200,v300,z1,TCP\WObj:=Workobject_6;
        MoveL Target_8210,v300,z1,TCP\WObj:=Workobject_6;
        MoveL Target_8220,v300,z1,TCP\WObj:=Workobject_6;
        MoveL Target_8230,v300,z1,TCP\WObj:=Workobject_6;
        MoveL Target_8240,v300,z1,TCP\WObj:=Workobject_6;
        MoveL Target_8250,v300,z1,TCP\WObj:=Workobject_6;
        MoveL Target_8260,v300,z1,TCP\WObj:=Workobject_6;
        MoveL Target_8270,v300,z1,TCP\WObj:=Workobject_6;
        MoveL Target_8280,v300,z1,TCP\WObj:=Workobject_6;
        MoveL Target_8290,v300,z1,TCP\WObj:=Workobject_6;
        MoveL Target_8300,v300,z1,TCP\WObj:=Workobject_6;
        MoveL Target_8310,v300,z1,TCP\WObj:=Workobject_6;
        MoveL Target_8320,v300,z1,TCP\WObj:=Workobject_6;
        MoveL Target_8330,v300,z1,TCP\WObj:=Workobject_6;
        MoveL HOME,v300,z1,TCP\WObj:=Workobject_5;
    ENDPROC
    PROC Path_30()
        MoveJ Maintenance,v300,z1,TCP\WObj:=Workobject_5;
    ENDPROC
ENDMODULE
